// Mitsubishi GX Works2 project: 化成2号柜-5.30   PLC: Q03UDE
// 化成线2号柜

TYPE BarCylinderIO : STRUCT
  xPresentSwitch : BOOL;  (* 行程开关 *)
  xBarCylinder : BOOL;  (* 阻挡气缸 *)
  xEmpty : BOOL;  (* 为空指示 *)
  xTransportMotorCW : BOOL;  (* 输送电机正转 *)
  tLeaveDelay : TIME;  (* 放行延时 *)
  xUnload : BOOL;  (* 下料 *)
  xBarCylinderButton : BOOL;  (* 阻挡气缸 *)
  xTransportMotorCWButton : BOOL;  (* 输送电机正转按钮 *)
  xLoad : BOOL;  (* 上料 *)
  xNextRun : BOOL;  (* 下位设备开始运行 *)
  xTransportMotorCCWButton : BOOL;  (* 输送电机反转按钮 *)
  xTransportMotorCCW : BOOL;  (* 输送电机反转 *)
END_STRUCT END_TYPE

TYPE ConveyorIO : STRUCT
  xCWPresent : BOOL;  (* 正转检测有无传感器 *)
  xCCWPresent : BOOL;  (* 反转检测有无传感器 *)
  xLoad : BOOL;  (* 上料请求 *)
  xUnload : BOOL;  (* 下料请求 *)
  xMotorCW : BOOL;  (* 电机正转 *)
  xMotorCCW : BOOL;  (* 电机反转 *)
  xEmpty : BOOL;  (* 线体状态为空 *)
  xNextRun : BOOL;  (* 下段线体运行 *)
  xUnloadCCW : BOOL;  (* 下料为反转 *)
  xloadCCW : BOOL;  (* 上料为反转 *)
  xLeave : BOOL;  (* 已经离开 *)
  xForward : BOOL;  (* 正转手动 *)
  xBackward : BOOL;  (* 反转手动 *)
  xBusy : BOOL;  (* 工作中 *)
  xPutInto : BOOL;  (* 线体直接投入物料 *)
  xUnloadAlarm : BOOL;  (* 下料报警 *)
  tLoadDelay : TIME;  (* 进入延时设置 *)
  xPosLimit : BOOL;  (* 正限位 *)
  xNegLimit : BOOL;  (* 负限位 *)
  xOverWidthAlarm : BOOL;  (* 超宽报警 *)
  xLimitAlarrm : BOOL;  (* 限位报警 *)
  iDeviceID : INT;  (* 线体ID *)
END_STRUCT END_TYPE

TYPE RGVCommunication : STRUCT
  xFullLoadRequest : BOOL;  (* 满框上料请求 *)
  xFullUnloadRequest : BOOL;  (* 满框下料请求 *)
  xEmptyLoadRequest : BOOL;  (* 空框上料请求 *)
  xEmptyUnloadRequest : BOOL;  (* 空框下料请求 *)
  xFullLoadRequestAkn : BOOL;  (* 满框上料请求确认 *)
  xFullUnloadRequestAkn : BOOL;  (* 满框下料请求确认 *)
  xEmptyLoadRequestAkn : BOOL;  (* 空框上料请求确认 *)
  xEmptyUnloadRequestAkn : BOOL;  (* 空框下料请求确认 *)
  xFullLoadComplete : BOOL;  (* 满框上料完成 *)
  xFullUnloadComplete : BOOL;  (* 满框下料完成 *)
  xEmptyLoadComplete : BOOL;  (* 空框上料完成 *)
  xEmptyUnloadComplete : BOOL;  (* 空框下料完成 *)
  xFullLoadCompleteAkn : BOOL;  (* 满框上料完成确认 *)
  xFullUnloadCompleteAkn : BOOL;  (* 满框下料完成确认 *)
  xEmptyLoadCompleteAkn : BOOL;  (* 空框上料完成确认 *)
  xEmptyUnloadCompleteAkn : BOOL;  (* 空框下料完成确认 *)
  iCurrentPostion : INT;  (* RGV当前位置 *)
  iDestinationPos : INT;  (* RGV目标位置 *)
  xMdiExe : BOOL;  (* RGV 执行 *)
  xMdiDone : BOOL;  (* RGV 执行完成 *)
  xEmpty1 : BOOL;
  xNextRun1 : BOOL;
  xEmpty2 : BOOL;
  xNextRun2 : BOOL;
  xLoad1 : BOOL;
  xUnload1 : BOOL;
  xLoad2 : BOOL;
  xUnload2 : BOOL;
  xCollisionAlarm : BOOL;  (* 干涉报警 *)
  xRemoteReset : BOOL;  (* 远程复位 *)
  xAuto : BOOL;  (* 自动 *)
END_STRUCT END_TYPE

TYPE ShuttleCarIO : STRUCT
  xReady : BOOL;  (* 准备就绪 *)
  xForward : BOOL;  (* 正转 *)
  xBackward : BOOL;  (* 反转 *)
  iCurrentPos : INT;  (* 当前位置 *)
  iDestinationPos : INT;  (* 目标位置 *)
  xCW : BOOL;  (* 正转输出 *)
  xCCW : BOOL;  (* 反转输出 *)
  xBrake : BOOL;  (* 刹车 *)
  xHomeSwitch : BOOL;  (* 零位接近开关 *)
  xPosLimit : BOOL;  (* 正限位 *)
  xNegLimit : BOOL;  (* 负限位 *)
  xMDIExe : BOOL;  (* MDI开始 *)
  xMDIDone : BOOL;  (* MDI 完成 *)
  xPassLimit : BOOL;  (* 限位屏蔽 *)
  xPosLimitCatch : BOOL;  (* 正限位捕捉 *)
  xNegLimitCatch : BOOL;  (* 负限位捕捉 *)
  xHomeExe : BOOL;  (* 开始寻零 *)
  xHomeDone : BOOL;  (* 寻零完成 *)
  xHomeBusy : BOOL;  (* 寻零中 *)
  xHomeFailed : BOOL;  (* 寻零失败 *)
  xBusy : BOOL;  (* 工作中 *)
  tArriveDelay : TIME;  (* 到位延时 *)
  xCylinder : BOOL;  (* 气缸控制 *)
  tBrakeDelay : TIME;  (* 抱闸延时 *)
  xPauseRamp : BOOL;  (* 暂停减速斜坡标志位 *)
  xPresentDetect1 : BOOL;  (* 物料有无检测1 *)
  xPresentDetect2 : BOOL;  (* 物料有无检测2 *)
  xOvertimeAlarm : BOOL;  (* 超时报警 *)
  tSetOverTime : TIME;  (* 设置超时时间 *)
  xLooseDetect : BOOL;  (* 松绳检测 *)
  xLooseAlarm : BOOL;  (* 松绳报警 *)
END_STRUCT END_TYPE

TYPE SwitchIO : STRUCT
  xLiftCylinderRetractDetect : BOOL;
  xLiftCylinderExtendDetect : BOOL;
  xLiftCylinderRetract : BOOL;
  xLiftCylinderExtend : BOOL;
  xEntryBarCylinderRetract : BOOL;
  xLiftCylinderExtendInit : BOOL;
  xEntryEnable : BOOL;
  xExitEnable : BOOL;
  xExitBarCylinderRetract : BOOL;
  xSwithEnable : BOOL;
  xLiftCylinderRetractButton : BOOL;
  xLiftCylinderExtendButton : BOOL;
  xEntryBarCylinderRetractButton : BOOL;
  xExitBarCylinderRetractButton : BOOL;
END_STRUCT END_TYPE

TYPE Stub : STRUCT
  xLoadRequest : BOOL;
  xLoadRequestAkn : BOOL;
  xUnloadRequest : BOOL;
  xUnloadRequestAkn : BOOL;
END_STRUCT END_TYPE

TYPE AccumulateConveyorIO : STRUCT
  xBarCylinderButton : BOOL;  (* 阻挡气缸按钮 *)
  xBarCylinder : BOOL;  (* 阻挡气缸 *)
  xLoad : BOOL;  (* 上料 *)
  xEmpty : BOOL;  (* 为空指示 *)
  xNextRun : BOOL;  (* 下位设备开始运行 *)
  xUnload : BOOL;  (* 下料 *)
  xTransportMotorCWButton : BOOL;  (* 输送电机正转按钮 *)
  xTransportMotorCW : BOOL;  (* 输送电机正转 *)
  xTransportMotorCCWButton : BOOL;  (* 输送电机反转按钮 *)
  xTransportMotorCCW : BOOL;  (* 输送电机反转 *)
  tLeaveDelay : TIME;  (* 放行延时 *)
  xPresentSwitch : BOOL;  (* 行程开关正向 *)
  xPresentSwitchEntry : BOOL;  (* 行程开关反向 *)
  xBarCylinderSecondary : BOOL;  (* 阻挡第二个无料的气缸 *)
  xBarSecondaryButton : BOOL;  (* 阻挡第二个无料的气缸手动按钮 *)
  xTwoWay : BOOL;  (* 双向积放线 *)
  iAccumulate : INT;  (* 数量 *)
  xLoadDone : BOOL;  (* 上料完成 *)
  tLoadDelay : TIME;  (* 上料延时 *)
  iDeviceID : INT;
END_STRUCT END_TYPE

// global labels: Global1
VAR_GLOBAL
  g_xAuto AT M11 : BOOL;  (* 自动 *)
  g_xManual : BOOL;  (* 手动 *)
  g_xEStop AT X3 : BOOL;  (* 急停 *)
  g_xReset AT X0 : BOOL;  (* 复位 *)
  g_xStackLampRed AT Y100 : BOOL;
  g_xStackLampAmber AT Y101 : BOOL;
  g_xStackLampGreen AT Y102 : BOOL;
  g_xBuzzer AT Y103 : BOOL;
  g_xStop AT M2 : BOOL;  (* 停止 *)
  g_xLocalAutoStart AT M1 : BOOL;  (* 本地自动启动 *)
  g_xRemoteAutoStart AT M0 : BOOL;  (* 远程自动启动 *)
  g_xRemoteAuto AT M10 : BOOL;  (* 远程 *)
  g_iState AT D40 : INT;  (* 当前状态 *)
  g_iLocalAutoStep : INT;
  g_xError : BOOL;
  g_xStart : BOOL;  (* 启动 *)
  g_xResetSingle AT M4 : BOOL;  (* 单线体复位 *)
  g_iDeviceIDSelect AT D0 : INT;  (* 线体编号选择 *)
  g_xPause AT M3 : BOOL;  (* 暂停 *)
  g_xAlarm : BOOL;  (* 报警 *)
  g_xInsertTask AT M5 : BOOL;  (* 单线体插入 *)
  g_iInsertTask AT D2 : INT;  (* 插入数据 *)
END_VAR

// global labels: Global
VAR_GLOBAL
  g_xQuarPackageRGVComFailed : BOOL;
  g_xChemRGVComFailed : BOOL;
  g_xChem1ComFailed : BOOL;
END_VAR

// task Task_01 (event TRUE, interval 0, priority 31): Start, POU, UDP

FUNCTION_BLOCK BarCylinder
VAR_IN_OUT
  BarCylinderIO : BarCylinderIO;
END_VAR
VAR
  m_tonViaDelay : TON;  (* 卸料延时定时器 *)
  m_xViaDelay : BOOL;  (* 通过延时 *)
  m_tViaDelayElapse : TIME;  (* 通过延时当前时间 *)
  m_xInitial : BOOL;  (* 初始化 *)
END_VAR
  (***********************************************************************
阻挡器模块，
由一个行程开关，一个阻挡器，一个倍速链输送电机组成
具有手动与自动模式
xEmpty显示当前为空料的状态
xUnload为卸料信号，连接下一设备的xEmpty信号
*************************************************************************)

  (*初始化，离开延时时间设置为5秒*)
IF NOT m_xInitial THEN
	 BarCylinderIO.tLeaveDelay :=T#5s;
	m_xInitial:=1;
END_IF;
IF g_xManual THEN    (*手动*)
	BarCylinderIO.xNextRun:=0;
	IF BarCylinderIO.xBarCylinderButton THEN
		BarCylinderIO.xBarCylinder:=1;
	ELSE
		BarCylinderIO.xBarCylinder:=0;
	END_IF;
	IF BarCylinderIO.xTransportMotorCWButton 
		AND NOT BarCylinderIO.xTransportMotorCCWButton 
		AND NOT BarCylinderIO.xTransportMotorCCW   THEN
		BarCylinderIO.xTransportMotorCW:=1;
	ELSE
		BarCylinderIO.xTransportMotorCW:=0;
	END_IF;
	IF BarCylinderIO.xTransportMotorCCWButton 
		AND NOT BarCylinderIO.xTransportMotorCWButton 
		AND NOT BarCylinderIO.xTransportMotorCW   THEN
		BarCylinderIO.xTransportMotorCCW:=1;
	ELSE
		BarCylinderIO.xTransportMotorCCW:=0;
	END_IF;
END_IF;
(*离开延时定时器*)
m_tonViaDelay(IN:=NOT  BarCylinderIO.xPresentSwitch AND g_xAuto  ,PT:= BarCylinderIO.tLeaveDelay ,Q:= BarCylinderIO.xEmpty ,ET:=m_tViaDelayElapse );

IF g_xAuto THEN(*自动*)
    IF BarCylinderIO.xUnload  AND NOT BarCylinderIO.xEmpty AND NOT BarCylinderIO.xNextRun THEN(*收到卸料命令，当阻挡器不为空时*)
    	BarCylinderIO.xBarCylinder:=1;
    	BarCylinderIO.xNextRun:=1;(*确保下料命令只执行一次，防止物料在输送过程中又有卸料命令导致多事卸料*)
    	BarCylinderIO.xTransportMotorCW:=1;
    END_IF;
    IF NOT  BarCylinderIO.xUnload  THEN
    	BarCylinderIO.xNextRun:=0;
    END_IF;
    (*如果为空，气缸顶起*)
   IF  BarCylinderIO.xEmpty  THEN
   	   BarCylinderIO.xBarCylinder:=0;
   	   IF BarCylinderIO.xLoad THEN
	   	   BarCylinderIO.xTransportMotorCW:=1;
	   END_IF;
   END_IF;
   IF NOT BarCylinderIO.xUnload AND NOT  BarCylinderIO.xEmpty THEN
   	    BarCylinderIO.xTransportMotorCW:=0;
   	END_IF;
END_IF;
IF NOT g_xEStop THEN
	 BarCylinderIO.xTransportMotorCW:=0;
	 BarCylinderIO.xTransportMotorCCW:=0;
	 BarCylinderIO.xBarCylinder:=0;
END_IF;
END_FUNCTION_BLOCK

FUNCTION_BLOCK Conveyor
VAR
  tRundelay : TIME;  (* 离开延时 *)
END_VAR
VAR_IN_OUT
  ConveyorMotor : ConveyorIO;  (* 输送线输入输出 *)
END_VAR
VAR
  iStep : INT;  (* 上料步骤 *)
  m_tUnloadTimer : TIME;  (* 下料计时器 *)
  m_tonLeaveDelay : TON;  (* 离开延时定时器 *)
  m_xLeaveDelayOut : BOOL;  (* 离开延时 *)
  m_tLeaveCurrentTime : TIME;
END_VAR
VAR CONSTANT
  LOAD_UNLOAD_TIME : TIME := T#30s;  (* 延时报警常量 *)
END_VAR
VAR
  m_tonUnloadAlam : TON;  (* 下料报警定时器 *)
  m_tonLoadDelay : TON;  (* 离开延时定时器 *)
  m_xLoadDelayOut : BOOL;  (* 离开延时 *)
  m_tLoadCurrentTime : TIME;
  m_xInitial : BOOL;  (* 初始化 *)
  m_tLoadTimer : TIME;  (* 上料延时当前时间 *)
END_VAR
(*////////////////////////////////////////////////////////////////////////////////////////////////////////////
//传输线控制FB块，可控制单方向线体，双向旋转线体，支持双向上下料            
//线体初始化后为空的情况下输入xLoad信号即可进行上料动作，使用xLoadCCW信号可反方向上料
//增加了产品信息和产品种类的储存，当传输线为空和上料进行标志位为零的情况下清除产品信息和产品种类
//使用方式是在置位xLoad信号后，把产品信息和产品种类传入，等下料后自动清零
//线体不为空的情况下使用xUnload信号可进行下料动作，物料有无传感器的下降沿后出发计时器，延时断开传输线旋转
//单方向传输线体把xLoadCCW、xUnloadCCW设置为零，双向线体上料方向和下料反向的,方向固定的 把xUnloadCCW设置为1
//双方向线体双向都能上下料的要根据上料的方向来设置xLoadCCW,xUnloadCCW
//增加工作中信号xBusy当电机正转 显示为工作中
//增加上下料超时报警，xLoadAlarm，xUnloadAlarm，设定时间在LOAD_UNLOAD_TIME常量上，现在设置的为30秒
//增加xPutInto信号，用于直接投入的物料，检测开关感应到后，直接进入下料流程，上升沿有效
//离开延时改为变量 iLeaveDelay 默认为0 离开检测开关离输送线尾端比较远的线体需要根据情况设定100ms为单位
增加初始化标志位，增加进入延时时间，初始化为进入延时时间为0 ，离开延时时间为2S，通过外围接口可以更改
//修改信息  修改后请增加版本
//YAO      V1.0
///////////////////////////////////////////////////////////////////////////////////////////////////////////
********************************************************)
IF NOT m_xInitial THEN
	ConveyorMotor.tLoadDelay:=T#100ms;
	ConveyorMotor.xNegLimit:=1;
	ConveyorMotor.xPosLimit:=1;
END_IF;
m_xInitial:=1;
IF g_xAuto THEN
CASE iStep OF
	0:
	ConveyorMotor.xMotorCW:=0;
	ConveyorMotor.xMotorCCW:=0;
	ConveyorMotor.xNextRun:=0;
IF g_xEStop AND NOT ConveyorMotor.xLimitAlarrm  THEN
	IF (ConveyorMotor.xCWPresent OR ConveyorMotor.xCCWPresent)  THEN
		iStep:=3;
		ConveyorMotor.xEmpty:=0;
		ELSE
		iStep:=1;
		ConveyorMotor.xEmpty:=1;
	END_IF;
END_IF;		
	1: 
	IF ConveyorMotor.xLoad    
		AND ConveyorMotor.xMotorCW=0   
		AND ConveyorMotor.xMotorCCW=0   
		AND ConveyorMotor.xEmpty THEN	
		iStep:=2;
	END_IF;
	2: 
	IF ConveyorMotor.xloadCCW THEN
		ConveyorMotor.xMotorCCW:=1; 
		ConveyorMotor.xMotorCW:=0;
	ELSE
	    ConveyorMotor.xMotorCW:=1;  
		ConveyorMotor.xMotorCCW:=0;
	END_IF;
		m_tonLoadDelay(IN:= (ConveyorMotor.xCWPresent AND NOT ConveyorMotor.xloadCCW) 
		                                        OR (ConveyorMotor.xCCWPresent AND ConveyorMotor.xloadCCW) ,
		                               PT:= ConveyorMotor.tLoadDelay ,
		                               Q:= m_xLoadDelayOut ,
		                               ET:= m_tLoadTimer );
	    IF m_xLoadDelayOut THEN 	 
		    iStep:=3;
		END_IF;
	3:
	ConveyorMotor.xMotorCW:=0;
	ConveyorMotor.xMotorCCW:=0;
	ConveyorMotor.xEmpty:=0;
	IF ConveyorMotor.xUnload AND NOT ConveyorMotor.xOverWidthAlarm THEN 
		iStep:=4;
	END_IF;
	4:	
	IF ConveyorMotor.xUnloadCCW THEN   
		ConveyorMotor.xMotorCCW:=1;  
		ConveyorMotor.xMotorCW:=0;
		ELSE
	    ConveyorMotor.xMotorCW:=1;  
		ConveyorMotor.xMotorCCW:=0;
	END_IF;
	ConveyorMotor.xNextRun:=1; 
	IF NOT ConveyorMotor.xUnload THEN 
		istep:=0;
	END_IF;
END_CASE;
IF LDP(TRUE,ConveyorMotor.xPutInto) THEN
	iStep:=0;
END_IF;
END_IF;
IF g_xManual THEN
	iStep:=0;

	IF ConveyorMotor.xForward 
		AND ConveyorMotor.xBackward=0 
		AND ConveyorMotor.xMotorCCW=0
		AND g_xEStop THEN
		ConveyorMotor.xMotorCW:=1;
		ConveyorMotor.xMotorCCW:=0;
		ELSE
		ConveyorMotor.xMotorCW:=0;
	END_IF;

	IF ConveyorMotor.xBackward 
		AND ConveyorMotor.xForward=0 
		AND ConveyorMotor.xMotorCW=0
		AND g_xEStop  THEN
		ConveyorMotor.xMotorCCW:=1;
		conveyormotor.xMotorCW:=0;
		ELSE
		ConveyorMotor.xMotorCCW:=0;
	END_IF;
END_IF;
IF ConveyorMotor.xMotorCCW        
	OR ConveyorMotor.xMotorCW THEN  
	ConveyorMotor.xBusy:=1;
	ELSE
	ConveyorMotor.xBusy:=0;
END_IF;
m_tonUnloadAlam(IN:= iStep=4,PT:= LOAD_UNLOAD_TIME,Q:= ConveyorMotor.xUnloadAlarm,ET:= m_tUnloadTimer );
(*//复位*)
IF (*g_xReset OR*)
	 (g_xResetSingle AND ConveyorMotor.iDeviceID=g_iDeviceIDSelect)THEN (*AND ConveyorMotor.iDeviceID=g_iDeviceIDSelect  THEN*)  (* //非正常情况下切断xNextRun不会复位，通过这个标志位会出发报警*)(*增加单体复位*)
	iStep:=0;
	ConveyorMotor.xNextRun:=0; 
	ConveyorMotor.xLimitAlarrm:=0;
	ConveyorMotor.xOverWidthAlarm:=0;
END_IF;
IF iStep=3 AND (NOT ConveyorMotor.xNegLimit OR NOT ConveyorMotor.xPosLimit) THEN
	ConveyorMotor.xOverWidthAlarm:=1;
END_IF;
IF ( ((ConveyorMotor.xloadCCW AND NOT ConveyorMotor.xNegLimit)            (*反转上料，碰到负限位*)
	OR  ( NOT ConveyorMotor.xloadCCW AND NOT ConveyorMotor.xPosLimit)) (*正转上料，碰到正限位*)
    AND iStep=2) (*上料过程*)
    OR
   ( iStep=4 (*下料过程*)
	AND( (ConveyorMotor.xUnloadCCW AND NOT ConveyorMotor.xPosLimit)  
	OR (NOT ConveyorMotor.xUnloadCCW AND NOT ConveyorMotor.xNegLimit)))    
    THEN
    ConveyorMotor.xLimitAlarrm:=1;
    iStep:=0;
END_IF;
END_FUNCTION_BLOCK

PROGRAM POU
VAR
  Lifter3 : ShuttleCar;
  Lifter3IO : ShuttleCarIO;
  H3000Conveyor11 : Conveyor;
  H3000Conveyor11IO : ConveyorIO;
  H3000Conveyor12 : Conveyor;
  H3000Conveyor12IO : ConveyorIO;
  H3000Conveyor13 : Conveyor;
  H3000Conveyor13IO : ConveyorIO;
  H3000Conveyor14 : Conveyor;
  H3000Conveyor14IO : ConveyorIO;
  H3000Conveyor15 : Conveyor;
  H3000Conveyor15IO : ConveyorIO;
  H3000Conveyor16 : Conveyor;
  H3000Conveyor16IO : ConveyorIO;
  H3000Conveyor17 : Conveyor;
  H3000Conveyor17IO : ConveyorIO;
  H3000Conveyor18 : Conveyor;
  H3000Conveyor18IO : ConveyorIO;
  H3000Conveyor19 : Conveyor;
  H3000Conveyor19IO : ConveyorIO;
  H3000Conveyor20 : Conveyor;
  H3000Conveyor20IO : ConveyorIO;
  H3000Conveyor21 : Conveyor;
  H3000Conveyor21IO : ConveyorIO;
  H3000Conveyor22 : Conveyor;
  H3000Conveyor22IO : ConveyorIO;
  H2200Conveyor13 : Conveyor;
  H2200Conveyor13IO : ConveyorIO;
  H2200Conveyor14 : Conveyor;
  H2200Conveyor14IO : ConveyorIO;
  H2200Conveyor15 : Conveyor;
  H2200Conveyor15IO : ConveyorIO;
  H2200Conveyor16 : Conveyor;
  H2200Conveyor16IO : ConveyorIO;
  H2200Conveyor17 : Conveyor;
  H2200Conveyor17IO : ConveyorIO;
  H2200Conveyor18 : Conveyor;
  H2200Conveyor18IO : ConveyorIO;
  H2200Conveyor19 : Conveyor;
  H2200Conveyor19IO : ConveyorIO;
  H2200Conveyor20 : Conveyor;
  H2200Conveyor20IO : ConveyorIO;
  H2200Conveyor21 : Conveyor;
  H2200Conveyor21IO : ConveyorIO;
  H2200Conveyor22 : Conveyor;
  H2200Conveyor22IO : ConveyorIO;
  H1000Conveyor11 : Conveyor;
  H1000Conveyor11IO : ConveyorIO;
  H1000Conveyor12 : Conveyor;
  H1000Conveyor12IO : ConveyorIO;
  H1000Conveyor13 : Conveyor;
  H1000Conveyor13IO : ConveyorIO;
  H1000Conveyor14 : Conveyor;
  H1000Conveyor14IO : ConveyorIO;
  H1000Conveyor15 : Conveyor;
  H1000Conveyor15IO : ConveyorIO;
  H1000Conveyor16 : Conveyor;
  H1000Conveyor16IO : ConveyorIO;
  H1000Conveyor19 : Conveyor;
  H1000Conveyor19IO : ConveyorIO;
  H1000Conveyor20 : Conveyor;
  H1000Conveyor20IO : ConveyorIO;
  Conveyor3 : Conveyor;
  Conveyor3IO : ConveyorIO;
  Lifter4 : ShuttleCar;
  Lifter4IO : ShuttleCarIO;
  Conveyor4 : Conveyor;
  Conveyor4IO : ConveyorIO;
  Lifter5 : ShuttleCar;
  Lifter5IO : ShuttleCarIO;
  Conveyor5 : Conveyor;
  Conveyor5IO : ConveyorIO;
  H850Conveyor1 : Conveyor;
  H850Conveyor1IO : ConveyorIO;
  H850Conveyor2 : Conveyor;
  H850Conveyor2IO : ConveyorIO;
  H2200Conveyor1 : Conveyor;
  H2200Conveyor1IO : ConveyorIO;
  ShuttleCar1 : ShuttleCar;
  ShuttleCar1IO : ShuttleCarIO;
  ConveyorShuttleCar : Conveyor;
  ConveyorShuttleCarIO : ConveyorIO;
  H1000Rotor1 : ShuttleCar;
  H1000Rotor1IO : ShuttleCarIO;
  H1000Rotor2 : ShuttleCar;
  H1000Rotor2IO : ShuttleCarIO;
  H1000Rotor1Cylinder : ShuttleCar;
  H1000Rotor1CylinderIO : ShuttleCarIO;
  H1000Rotor2Cylinder : ShuttleCar;
  H1000Rotor2CylinderIO : ShuttleCarIO;
  H850Conveyor1Trans : Conveyor;  (* 二封设备入口接驳 *)
  H850Conveyor1IOTrans : ConveyorIO;  (* 二封设备入口接驳 *)
  H850Conveyor2Trans : Conveyor;  (* 二封设备入口接驳 *)
  H850Conveyor2IOTrans : ConveyorIO;  (* 二封设备入口接驳 *)
  H850Conveyor3Trans : Conveyor;  (* 二封设备入口接驳 *)
  H850Conveyor3IOTrans : ConveyorIO;  (* 二封设备入口接驳 *)
  H850Conveyor4Trans : Conveyor;  (* 二封设备入口接驳 *)
  H850Conveyor4IOTrans : ConveyorIO;  (* 二封设备入口接驳 *)
  H850Conveyor5Trans : Conveyor;  (* 二封设备入口接驳 *)
  H850Conveyor5IOTrans : ConveyorIO;  (* 二封设备入口接驳 *)
  H850Conveyor6Trans : Conveyor;  (* 二封设备入口接驳 *)
  H850Conveyor6IOTrans : ConveyorIO;  (* 二封设备入口接驳 *)
  H850Conveyor7Trans : Conveyor;  (* 二封设备入口接驳 *)
  H850Conveyor7IOTrans : ConveyorIO;  (* 二封设备入口接驳 *)
  H850Conveyor8Trans : Conveyor;  (* 二封设备入口接驳 *)
  H850Conveyor8IOTrans : ConveyorIO;  (* 二封设备入口接驳 *)
  Lifter4VelocityCtl : ShuttleCarVelocityFB;
  Lifter5VelocityCtl : ShuttleCarVelocityFB;
  m_tofShuttleCar1LeaveDelay : TOF;  (* f *)
  m_xShuttleCar1LeaveDelay : BOOL;
  m_tShuttleCar1LeaveDelay : TIME;
  Lifter3VelocityCtl : ShuttleCarVelocityFB;
  H380EmptyABumperBar : AccumulateConveyor;
  H380EmptyABumperBarIO : AccumulateConveyorIO;
  H380EmptyBBumperBar : AccumulateConveyor;
  H380EmptyBBumperBarIO : AccumulateConveyorIO;
  ChemRGV : RGVCommunication;
  QuarPackageRGV : RGVCommunication;
  m_iH1000Rotor2Step : INT;
  m_iH1000Rotor1Step : INT;
  QuarPackage1Stub : Stub;
  QuarPackage2Stub : Stub;
  QuarPackage3Stub : Stub;
  QuarPackage4Stub : Stub;
  Chem1Stub : Stub;
  Chem2Stub : Stub;
  Chem3Stub : Stub;
  Chem4Stub : Stub;
  Chem5Stub : Stub;
  Chem6Stub : Stub;
  Chem7Stub : Stub;
  Chem8Stub : Stub;
  Chem9Stub : Stub;
  Chem10Stub : Stub;
  Chem11Stub : Stub;
  Chem12Stub : Stub;
  m_tonXD8 : TON;
  m_xXD8 : BOOL;
  m_tXD8 : TIME;
  m_xXD8Lock : BOOL;
  m_xDirection : BOOL;  (* 空框方向信息 *)
  m_xRotor2Done : BOOL;  (* 上料转台旋转完成 *)
  m_xRotor1Done : BOOL;  (* 下料转台旋转完成 *)
  m_xRotor1Start : BOOL;  (* 下料转台旋转开始 *)
  m_xRotor2Start : BOOL;  (* 上料转台旋转开始 *)
  m_xDischargeAkn : BOOL;  (* 下料确认 *)
  m_xFomationRGVAuto : BOOL;
  m_xDebindCode : BOOL;
  m_xCheckDone : BOOL;  (* 品检完成 *)
  m_xAllCheck : BOOL;  (* 全检工位 *)
  m_xAllCheckOver : BOOL;  (* 全检完毕按钮 *)
  m_xPassAllow : BOOL;  (* 全检放行 *)
  m_arrxRGVEmptyTaskCondition : ARRAY [0..9] OF BOOL;  (* 空框回流任务 *)
  RGVEmptyTask : PriorityFB;
  m_iRGVEmptyTask : INT;
  H380EmptyBRotorConveyorIO : ConveyorIO;
  H380EmptyBLifter : ShuttleCar;  (* 空框B转台升降气缸 *)
  H380EmptyBLifterIO : ShuttleCarIO;
  H380EmptyBRotor : ShuttleCar;  (* 空框B转台 *)
  H380EmptyBRotorIO : ShuttleCarIO;
  m_xEmptyBRotorStart : BOOL;  (* 空框B旋转开始 *)
  m_xEmptyBRotorDone : BOOL;  (* 空框B旋转完毕 *)
  m_iEmptyBRotorStep : INT;  (* 空框B旋转步 *)
  m_xLoadDirection : BOOL;  (* 上料口方向信息 *)
  m_xUnloadDirection : BOOL;  (* 下料口方向信息 *)
  H380EmptyBRotorConveyor : Conveyor;  (* 空框B转台Conveyor *)
  H380EmptyARotorConveyor : Conveyor;  (* 空框A转台Conveyor *)
  H380EmptyARotorConveyorIO : ConveyorIO;
  H380EmptyALifter : ShuttleCar;  (* 空框A转台升降气缸 *)
  H380EmptyALifterIO : ShuttleCarIO;
  H380EmptyARotor : ShuttleCar;  (* 空框A转台 *)
  H380EmptyARotorIO : ShuttleCarIO;
  m_xEmptyARotorStart : BOOL;  (* 空框A旋转开始 *)
  m_xEmptyARotorDone : BOOL;  (* 空框A旋转完毕 *)
  m_iEmptyARotorStep : INT;  (* 空框A旋转步 *)
  TON_BRotorStep5 : TON;  (* 空框B转台第5步计时 *)
  m_xBRotorStep5 : BOOL;
  m_tBRotorStep5 : TIME;
  TON_ARotorStep5 : TON;  (* 空框A转台第5步延时 *)
  m_xARotorStep5 : BOOL;
  m_tARotorStep5 : TIME;
  H2200SudsecitonCylinderA3 : BarCylinder;  (* 空框回流A线3阻挡气缸 *)
  H2200SudsecitonCylinderA4 : BarCylinder;  (* 空框回流A线4阻挡气缸 *)
  H2200SudsecitonCylinderA5 : BarCylinder;  (* 空框回流A线5阻挡气缸 *)
  H2200SudsecitonCylinderA3IO : BarCylinderIO;  (* 空框回流A线3阻挡气缸 *)
  H2200SudsecitonCylinderA4IO : BarCylinderIO;  (* 空框回流A线4阻挡气缸 *)
  H2200SudsecitonCylinderA5IO : BarCylinderIO;  (* 空框回流A线5阻挡气缸 *)
  H2200SudsecitonCylinderB3 : BarCylinder;  (* 空框回流B线3阻挡气缸 *)
  H2200SudsecitonCylinderB4 : BarCylinder;  (* 空框回流B线4阻挡气缸 *)
  H2200SudsecitonCylinderB5 : BarCylinder;  (* 空框回流B线5阻挡气缸 *)
  H2200SudsecitonCylinderB3IO : BarCylinderIO;  (* 空框回流B线3阻挡气缸 *)
  H2200SudsecitonCylinderB4IO : BarCylinderIO;  (* 空框回流B线4阻挡气缸 *)
  H2200SudsecitonCylinderB5IO : BarCylinderIO;  (* 空框回流B线5阻挡气缸 *)
  m_tonSudsecitonCylinderA3Delay : TON;  (* 空框回流A线5阻挡气缸 *)
  m_tCylinderA3DelayCurrentTime : TIME;
  m_tonSudsecitonCylinderA4Delay : TON;
  m_tCylinderA4DelayCurrentTime : TIME;
  m_tonSudsecitonCylinderA5Delay : TON;
  m_tCylinderA5DelayCurrentTime : TIME;
  m_tonSudsecitonCylinderB3Delay : TON;
  m_tCylinderB3DelayCurrentTime : TIME;
  m_tonSudsecitonCylinderB4Delay : TON;
  m_tCylinderB4DelayCurrentTime : TIME;
  m_tonSudsecitonCylinderB5Delay : TON;
  m_tCylinderB5DelayCurrentTime : TIME;
  BlockA : BOOL;  (* 空框回流A线阻塞 *)
  BlockB : BOOL;  (* 空框回流B线阻塞 *)
END_VAR
(*---------我在516行加了一整行*)
Lifter3(ShuttleCarInOut:=Lifter3IO);
ShuttleCarCurrentPosition( X5A OR X5B ,X5A ,X5B, FALSE, Lifter3IO.iCurrentPos );
Lifter3VelocityCtl(xEnable:= g_xManual,xMotorCW:= Lifter3IO.xCW ,xMotorCCW:= Lifter3IO.xCCW ,
                               xPosition1Switch:= X5A ,xDecelerationSwitch:= X59 ,
	                           xPosition2Switch:=X5B ,xHighSpeed:= Y163);
Lifter3IO.xReady:=X4;
Lifter3Io.xForward:=M50;
Lifter3IO.xBackward:=M51;
Lifter3IO.xPosLimit:=X5C;
Lifter3IO.xNegLimit:=X5D;
Lifter3Io.xLooseDetect:=X5E;
M130:=Lifter3IO.xLooseDetect;
Y161:=Lifter3IO.xCW;
Y162:=Lifter3IO.xCCW;
Y166:=Lifter3IO.xBrake;

Conveyor3(ConveyorMotor:=Conveyor3IO);
Conveyor3IO.xForward:=M52;
Conveyor3IO.xBackward:=M53;
Conveyor3IO.xCWPresent:=X61;
Conveyor3IO.xCCWPresent:=X62;
Y168:=Conveyor3IO.xMotorCW;
Y167:=Conveyor3IO.xMotorCCW;
Conveyor3IO.xUnloadCCW:=1;
Conveyor3IO.iDeviceID:=3;

Lifter4(ShuttleCarInOut:=Lifter4IO);
ShuttleCarCurrentPosition( X64 OR X65 ,X64 ,X65, FALSE, Lifter4IO.iCurrentPos );
Lifter4VelocityCtl(xEnable:= g_xAuto,xMotorCW:= Lifter4IO.xCW ,xMotorCCW:= Lifter4IO.xCCW ,
                               xPosition1Switch:= X64 ,xDecelerationSwitch:= X63 ,
	                           xPosition2Switch:=X65 ,xHighSpeed:= Y16B);
Lifter4IO.xReady:=X5;
Lifter4Io.xForward:=M54;
Lifter4IO.xBackward:=M55;
Lifter4IO.xPosLimit:=X66;
Lifter4IO.xNegLimit:=X67;
Lifter4IO.xLooseDetect:=X68;
M129:=Lifter4IO.xLooseAlarm;
Y169:=Lifter4IO.xCW;
Y16A:=Lifter4IO.xCCW;
Y16E:=Lifter4IO.xBrake;

Conveyor4(ConveyorMotor:=Conveyor4IO);
Conveyor4IO.xForward:=M56;
Conveyor4IO.xBackward:=M57;
Conveyor4IO.xCWPresent:=X6B;
Conveyor4IO.xCCWPresent:=X6C;
Y170:=Conveyor4IO.xMotorCW;
Y16F:=Conveyor4IO.xMotorCCW;
Conveyor4IO.xUnloadCCW:=1;
Conveyor4IO.iDeviceID:=4;

Lifter5(ShuttleCarInOut:=Lifter5IO);
ShuttleCarCurrentPosition( X6E OR X6F ,X6E ,X6F, FALSE, Lifter5IO.iCurrentPos );
Lifter5VelocityCtl(xEnable:= g_xAuto,
                               xMotorCW:= Lifter5IO.xCW ,
                               xMotorCCW:= Lifter5IO.xCCW,
                               xPosition1Switch:=X6E,
                               xDecelerationSwitch:= X6D,
	                           xPosition2Switch:=X6F,
	                           xHighSpeed:= Y173 );
Lifter5IO.xReady:=X6;
Lifter5Io.xForward:=M58;
Lifter5IO.xBackward:=M59;
Lifter5IO.xPosLimit:=X70;
Lifter5IO.xNegLimit:=X71;
Lifter5IO.xLooseDetect:=X72;
M128:=Lifter5IO.xLooseAlarm;
Y171:=Lifter5IO.xCW;
Y172:=Lifter5IO.xCCW;
Y176:=Lifter5IO.xBrake;

Conveyor5(ConveyorMotor:=Conveyor5IO);
Conveyor5IO.xForward:=M60;
Conveyor5IO.xBackward:=M61;
Conveyor5IO.xCWPresent:=X75;
Conveyor5IO.xCCWPresent:=X76;
Y178:=Conveyor5IO.xMotorCW;
Y177:=Conveyor5IO.xMotorCCW;
Conveyor5IO.xUnloadCCW:=1;
Conveyor5IO.iDeviceID:=5;

ShuttleCar1(ShuttleCarInOut:=ShuttleCar1IO);
ShuttleCarCurrentPosition(( NOT X53 AND NOT X54) OR (NOT X53 AND NOT X55) OR (NOT X54 AND NOT  X55) ,
                                                       NOT X53 AND NOT X54 ,
                                                       NOT X53 AND NOT X55,
                                                       NOT X54 AND NOT  X55, 
                                                       ShuttleCar1IO.iCurrentPos );
ShuttleCar1IO.xReady:=X7;
ShuttleCar1IO.xForward:=M62;
ShuttleCar1IO.xBackward:=M63;
ShuttleCar1IO.xPosLimit:=X51;
ShuttleCar1IO.xNegLimit:=X52;
Y1AC:=ShuttleCar1IO.xCW;
Y1AB:=ShuttleCar1IO.xCCW;
Y12B:=ShuttleCar1IO.xBrake;

ConveyorShuttleCar(ConveyorMotor:=ConveyorShuttleCarIO);
ConveyorShuttleCarIO.xForward:=M64;
ConveyorShuttleCarIO.xBackward:=M65;
ConveyorShuttleCarIO.xCWPresent:=X56;
ConveyorShuttleCarIO.xCCWPresent:=X57;
Y153:=ConveyorShuttleCarIO.xMotorCW;
Y154:=ConveyorShuttleCarIO.xMotorCCW;
ConveyorShuttleCarIO.iDeviceID:=6;

H3000Conveyor11(ConveyorMotor:=H3000Conveyor11IO);
H3000Conveyor11IO.xForward:=M30;
H3000Conveyor11IO.xCWPresent:=X8;
Y108:=H3000Conveyor11IO.xMotorCW;
H3000Conveyor11IO.iDeviceID:=3011;

H3000Conveyor12(ConveyorMotor:=H3000Conveyor12IO);
H3000Conveyor12IO.xForward:=M31;
H3000Conveyor12IO.xCWPresent:=X9;
Y109:=H3000Conveyor12IO.xMotorCW;
H3000Conveyor12IO.iDeviceID:=3012;

H3000Conveyor13(ConveyorMotor:=H3000Conveyor13IO);
H3000Conveyor13IO.xForward:=M32;
H3000Conveyor13IO.xCWPresent:=XA;
Y10A:=H3000Conveyor13IO.xMotorCW;
H3000Conveyor13IO.iDeviceID:=3013;

H3000Conveyor14(ConveyorMotor:=H3000Conveyor14IO);
H3000Conveyor14IO.xForward:=M33;
H3000Conveyor14IO.xCWPresent:=XB;
Y10B:=H3000Conveyor14IO.xMotorCW;
H3000Conveyor14IO.iDeviceID:=3014;

H3000Conveyor15(ConveyorMotor:=H3000Conveyor15IO);
H3000Conveyor15IO.xForward:=M34;
H3000Conveyor15IO.xCWPresent:=XC;
Y10C:=H3000Conveyor15IO.xMotorCW;
H3000Conveyor15IO.iDeviceID:=3015;

H3000Conveyor16(ConveyorMotor:=H3000Conveyor16IO);
H3000Conveyor16IO.xForward:=M34;
H3000Conveyor16IO.xCWPresent:=XD;
Y10D:=H3000Conveyor16IO.xMotorCW;
H3000Conveyor16IO.iDeviceID:=3016;

H3000Conveyor17(ConveyorMotor:=H3000Conveyor17IO);
H3000Conveyor17IO.xForward:=M35;
H3000Conveyor17IO.xCWPresent:=XE;
Y10E:=H3000Conveyor17IO.xMotorCW;
H3000Conveyor17IO.iDeviceID:=3017;

H3000Conveyor18(ConveyorMotor:=H3000Conveyor18IO);
H3000Conveyor18IO.xForward:=M36;
H3000Conveyor18IO.xCWPresent:=XF;
Y10F:=H3000Conveyor18IO.xMotorCW;
H3000Conveyor18IO.iDeviceID:=3018;

H3000Conveyor19(ConveyorMotor:=H3000Conveyor19IO);
H3000Conveyor19IO.xForward:=M37;
H3000Conveyor19IO.xCWPresent:=X10;
Y110:=H3000Conveyor19IO.xMotorCW;
H3000Conveyor19IO.iDeviceID:=3019;

H3000Conveyor20(ConveyorMotor:=H3000Conveyor20IO);
H3000Conveyor20IO.xForward:=M38;
H3000Conveyor20IO.xCWPresent:=X11;
Y111:=H3000Conveyor20IO.xMotorCW;
H3000Conveyor20IO.iDeviceID:=3020;

H3000Conveyor21(ConveyorMotor:=H3000Conveyor21IO);
H3000Conveyor21IO.xForward:=M39;
H3000Conveyor21IO.xCWPresent:=X12;
Y112:=H3000Conveyor21IO.xMotorCW;
H3000Conveyor21IO.iDeviceID:=3021;

H3000Conveyor22(ConveyorMotor:=H3000Conveyor22IO);
H3000Conveyor22IO.xForward:=M40;
H3000Conveyor22IO.xCWPresent:=X13;
Y113:=H3000Conveyor22IO.xMotorCW;
H3000Conveyor22IO.xNegLimit:=X14;
M98:=H3000Conveyor22IO.xOverWidthAlarm;
M99:=H3000Conveyor22IO.xLimitAlarrm;
H3000Conveyor22IO.iDeviceID:=3022;

H850Conveyor1(ConveyorMotor:=H850Conveyor1IO);
H850Conveyor1IO.xForward:=M41;
H850Conveyor1IO.xCWPresent:=X4E;
Y14E:=H850Conveyor1IO.xMotorCW;
H850Conveyor1IO.iDeviceID:=8501;

H850Conveyor2(ConveyorMotor:=H850Conveyor2IO);
H850Conveyor2IO.xForward:=M42;
H850Conveyor2IO.xCWPresent:=X4F;
Y14F:=H850Conveyor2IO.xMotorCW;
H850Conveyor2IO.iDeviceID:=8502;

H2200Conveyor1(ConveyorMotor:=H2200Conveyor1IO);
H2200Conveyor1IO.xForward:=M43;
H2200Conveyor1IO.xCWPresent:=X4D;
Y14D:=H2200Conveyor1IO.xMotorCW;
H2200Conveyor1IO.iDeviceID:=2201;


H2200Conveyor13(ConveyorMotor:=H2200Conveyor13IO);
H2200Conveyor13IO.xForward:=M44;
H2200Conveyor13IO.xCWPresent:=X2F;
Y12F:=H2200Conveyor13IO.xMotorCW;
H2200Conveyor13IO.iDeviceID:=2213;

H2200Conveyor14(ConveyorMotor:=H2200Conveyor14IO);
H2200Conveyor14IO.xForward:=M45;
H2200Conveyor14IO.xCWPresent:=X30;
Y130:=H2200Conveyor14IO.xMotorCW;
H2200Conveyor14IO.iDeviceID:=2214;

H2200Conveyor15(ConveyorMotor:=H2200Conveyor15IO);
H2200Conveyor15IO.xForward:=M46;
H2200Conveyor15IO.xCWPresent:=X31;
Y131:=H2200Conveyor15IO.xMotorCW;
H2200Conveyor15IO.iDeviceID:=2215;

H2200Conveyor16(ConveyorMotor:=H2200Conveyor16IO);
H2200Conveyor16IO.xForward:=M47;
H2200Conveyor16IO.xCWPresent:=X32;
Y132:=H2200Conveyor16IO.xMotorCW;
H2200Conveyor16IO.iDeviceID:=2216;

H2200Conveyor17(ConveyorMotor:=H2200Conveyor17IO);
H2200Conveyor17IO.xForward:=M48;
H2200Conveyor17IO.xCWPresent:=X33;
Y133:=H2200Conveyor17IO.xMotorCW;
H2200Conveyor17IO.iDeviceID:=2217;

H2200Conveyor18(ConveyorMotor:=H2200Conveyor18IO);
H2200Conveyor18IO.xForward:=M49;
H2200Conveyor18IO.xCWPresent:=X34;
Y134:=H2200Conveyor18IO.xMotorCW;
H2200Conveyor18IO.iDeviceID:=2218;

H2200Conveyor19(ConveyorMotor:=H2200Conveyor19IO);
H2200Conveyor19IO.xForward:=M70;
H2200Conveyor19IO.xCWPresent:=X35;
Y135:=H2200Conveyor19IO.xMotorCW;
H2200Conveyor19IO.iDeviceID:=2219;

H2200Conveyor20(ConveyorMotor:=H2200Conveyor20IO);
H2200Conveyor20IO.xForward:=M71;
H2200Conveyor20IO.xCWPresent:=X36;
Y136:=H2200Conveyor20IO.xMotorCW;
H2200Conveyor20IO.iDeviceID:=2220;

H2200Conveyor21(ConveyorMotor:=H2200Conveyor21IO);
H2200Conveyor21IO.xForward:=M72;
H2200Conveyor21IO.xCWPresent:=X37;
Y137:=H2200Conveyor21IO.xMotorCW;
H2200Conveyor21IO.iDeviceID:=2221;

H2200Conveyor22(ConveyorMotor:=H2200Conveyor22IO);
H2200Conveyor22IO.xForward:=M73;
H2200Conveyor22IO.xCWPresent:=X38;
Y138:=H2200Conveyor22IO.xMotorCW;
H2200Conveyor22IO.xNegLimit:=X15;
M118:=H2200Conveyor22IO.xOverWidthAlarm;
M119:=H2200Conveyor22IO.xLimitAlarrm;
H2200Conveyor22IO.iDeviceID:=2222;

H1000Conveyor11(ConveyorMotor:=H1000Conveyor11IO);
H1000Conveyor11IO.xForward:=M75;
H1000Conveyor11IO.xCWPresent:=X3A;
Y13A:=H1000Conveyor11IO.xMotorCW;
H1000Conveyor11IO.iDeviceID:=1011;

H1000Conveyor12(ConveyorMotor:=H1000Conveyor12IO);
H1000Conveyor12IO.xForward:=M76;
H1000Conveyor12IO.xCWPresent:=X3B;
Y13B:=H1000Conveyor12IO.xMotorCW;
H1000Conveyor12IO.iDeviceID:=1012;

H1000Conveyor13(ConveyorMotor:=H1000Conveyor13IO);
H1000Conveyor13IO.xForward:=M77;
H1000Conveyor13IO.xCWPresent:=X3C;
Y13C:=H1000Conveyor13IO.xMotorCW;
H1000Conveyor13IO.iDeviceID:=1013;

H1000Conveyor14(ConveyorMotor:=H1000Conveyor14IO);
H1000Conveyor14IO.xForward:=M78;
H1000Conveyor14IO.xCWPresent:=X3D;
Y13D:=H1000Conveyor14IO.xMotorCW;
H1000Conveyor14IO.iDeviceID:=1014;

H1000Conveyor15(ConveyorMotor:=H1000Conveyor15IO);
H1000Conveyor15IO.xForward:=M79;
H1000Conveyor15IO.xCWPresent:=X3E;
Y13E:=H1000Conveyor15IO.xMotorCW;
H1000Conveyor15IO.iDeviceID:=1015;

H1000Rotor2(ShuttleCarInOut:=H1000Rotor2IO);
ShuttleCarCurrentPosition( X9F OR X9E ,X9F ,X9E, FALSE, H1000Rotor2IO.iCurrentPos );
H1000Rotor2IO.xReady:=TRUE;
H1000Rotor2IO.xForward:=M93;
H1000Rotor2IO.xBackward:=M94;
H1000Rotor2IO.xPosLimit:=XB0;
H1000Rotor2IO.xNegLimit:=XB1;
Y1BC:=H1000Rotor2IO.xCW;
Y1BD:=H1000Rotor2IO.xCCW;
Y12A:=H1000Rotor2IO.xBrake;

H1000Rotor2Cylinder(ShuttleCarInOut:=H1000Rotor2CylinderIO);
ShuttleCarCurrentPosition( XA0 OR XA1 ,XA1 ,XA0, FALSE, H1000Rotor2CylinderIO.iCurrentPos );
H1000Rotor2CylinderIO.xReady:=TRUE;
H1000Rotor2CylinderIO.xForward:=M87;
H1000Rotor2CylinderIO.xBackward:=M88;
H1000Rotor2CylinderIO.xPosLimit:=TRUE;
H1000Rotor2CylinderIO.xNegLimit:=TRUE;
Y1A1:=H1000Rotor2CylinderIO.xCW;
Y1A0:=H1000Rotor2CylinderIO.xCCW;

H1000Conveyor16(ConveyorMotor:=H1000Conveyor16IO);
H1000Conveyor16IO.xForward:=M80;
H1000Conveyor16IO.xCWPresent:=X3F OR XC8;
Y13F:=H1000Conveyor16IO.xMotorCW;
H1000Conveyor16IO.iDeviceID:=1016;

H1000Rotor1(ShuttleCarInOut:=H1000Rotor1IO);
ShuttleCarCurrentPosition( X9A OR X9B ,X9A ,X9B, FALSE, H1000Rotor1IO.iCurrentPos );
H1000Rotor1IO.xReady:=TRUE;
H1000Rotor1IO.xForward:=M83;
H1000Rotor1IO.xBackward:=M84;
H1000Rotor1IO.xPosLimit:=X99;
H1000Rotor1IO.xNegLimit:=X98;
Y104:=H1000Rotor1IO.xCW;
Y105:=H1000Rotor1IO.xCCW;
Y129:=H1000Rotor1IO.xBrake;

H1000Rotor1Cylinder(ShuttleCarInOut:=H1000Rotor1CylinderIO);
ShuttleCarCurrentPosition( X9D OR X9C ,X9D ,X9C, FALSE, H1000Rotor1CylinderIO.iCurrentPos );
H1000Rotor1CylinderIO.xReady:=TRUE;
H1000Rotor1CylinderIO.xForward:=M85;
H1000Rotor1CylinderIO.xBackward:=M86;
H1000Rotor1CylinderIO.xPosLimit:=TRUE;
H1000Rotor1CylinderIO.xNegLimit:=TRUE;
Y19C:=H1000Rotor1CylinderIO.xCW;
Y19B:=H1000Rotor1CylinderIO.xCCW;

H1000Conveyor19(ConveyorMotor:=H1000Conveyor19IO);
H1000Conveyor19IO.xForward:=M81;
(*H1000Conveyor19IO.xCWPresent:=NOT X42;*)
H1000Conveyor19IO.xCWPresent:=XCE;
Y142:=H1000Conveyor19IO.xMotorCW;
H1000Conveyor19IO.xPosLimit:= X42;
(*H1000Conveyor19IO.xPosLimit:=1;*)
H1000Conveyor19IO.iDeviceID:=1019;
H1000Conveyor19IO.tLoadDelay:=T#200ms;
M138:=h1000Conveyor19IO.xLimitAlarrm;

H1000Conveyor20(ConveyorMotor:=H1000Conveyor20IO);
H1000Conveyor20IO.xForward:=M82;
H1000Conveyor20IO.xCWPresent:=X43;
Y143:=H1000Conveyor20IO.xMotorCW;
H1000Conveyor20IO.iDeviceID:=1020;

H850Conveyor1Trans(ConveyorMotor:=H850Conveyor1IOTrans);
H850Conveyor1IOTrans.xForward:=M120;
H850Conveyor1IOTrans.xCWPresent:=XA3;
Y1A3:=H850Conveyor1IOTrans.xMotorCW;
H850Conveyor1IOTrans.iDeviceID:=801;

H850Conveyor2Trans(ConveyorMotor:=H850Conveyor2IOTrans);
H850Conveyor2IOTrans.xForward:=M121;
H850Conveyor2IOTrans.xCWPresent:=XA4;
Y1A4:=H850Conveyor2IOTrans.xMotorCW;
H850Conveyor2IOTrans.iDeviceID:=802;

H850Conveyor3Trans(ConveyorMotor:=H850Conveyor3IOTrans);
H850Conveyor3IOTrans.xForward:=M122;
H850Conveyor3IOTrans.xCWPresent:=XA5;
Y1A5:=H850Conveyor3IOTrans.xMotorCW;
H850Conveyor3IOTrans.iDeviceID:=803;

H850Conveyor4Trans(ConveyorMotor:=H850Conveyor4IOTrans);
H850Conveyor4IOTrans.xForward:=M123;
H850Conveyor4IOTrans.xCWPresent:=XA6;
Y1A6:=H850Conveyor4IOTrans.xMotorCW;
H850Conveyor4IOTrans.iDeviceID:=804;

H850Conveyor5Trans(ConveyorMotor:=H850Conveyor5IOTrans);
H850Conveyor5IOTrans.xForward:=M124;
H850Conveyor5IOTrans.xCWPresent:=XA7;
Y1A7:=H850Conveyor5IOTrans.xMotorCW;
H850Conveyor5IOTrans.iDeviceID:=805;

H850Conveyor6Trans(ConveyorMotor:=H850Conveyor6IOTrans);
H850Conveyor6IOTrans.xForward:=M125;
H850Conveyor6IOTrans.xCWPresent:=XA8;
Y1A8:=H850Conveyor6IOTrans.xMotorCW;
H850Conveyor6IOTrans.iDeviceID:=806;

H850Conveyor7Trans(ConveyorMotor:=H850Conveyor7IOTrans);
H850Conveyor7IOTrans.xForward:=M126;
H850Conveyor7IOTrans.xCWPresent:=XA9;
Y1A9:=H850Conveyor7IOTrans.xMotorCW;
H850Conveyor7IOTrans.iDeviceID:=807;

H850Conveyor8Trans(ConveyorMotor:=H850Conveyor8IOTrans);
H850Conveyor8IOTrans.xForward:=M127;
H850Conveyor8IOTrans.xCWPresent:=XBA;
Y1AA:=H850Conveyor8IOTrans.xMotorCW;
H850Conveyor8IOTrans.iDeviceID:=808;

H380EmptyABumperBar( AccumulateConveyorIO:= H380EmptyABumperBarIO);
H380EmptyABumperBarIO.xBarCylinderButton:=M68;
H380EmptyABumperBarIO.xTransportMotorCWButton:=M89;
H380EmptyABumperBarIO.xTransportMotorCCWButton:=M90;
(*H380EmptyABumperBarIO.xPresentSwitch:=X48;*)
H380EmptyABumperBarIO.xPresentSwitchEntry:=X49;
Y148:=H380EmptyABumperBarIO.xBarCylinderSecondary OR M154;
Y149:=H380EmptyABumperBarIO.xBarCylinder OR M155;
Y15E:=H380EmptyABumperBarIO.xTransportMotorCW OR M156 ;(*往左为正转，下料方向为正*)
Y15D:=H380EmptyABumperBarIO.xTransportMotorCCW OR M157;
H380EmptyABumperBarIO.xTwoWay:=1;
H380EmptyABumperBarIO.tLoadDelay:=t#3S;
H380EmptyABumperBarIO.iDeviceID:=901;

H380EmptyARotorConveyor(ConveyorMotor:=H380EmptyARotorConveyorIO);
H380EmptyARotorConveyorIO.xCWPresent:=X7F;
H380EmptyARotorConveyorIO.xCCWPresent:=X7F;
H380EmptyARotorConveyorIO.tLoadDelay:=T#3S;
H380EmptyARotorConveyorIO.iDeviceID:=901;

H380EmptyALifter(ShuttleCarInOut:=H380EmptyALifterIO);(**升降**)
ShuttleCarCurrentPosition(  XC2 OR XC3 ,XC2 ,XC3,FALSE, H380EmptyALifterIO.iCurrentPos );
H380EmptyALifterIO.xReady:=TRUE;
H380EmptyALifterIO.xForward:=M26;
H380EmptyALifterIO.xBackward:=M27;
H380EmptyALifterIO.xPosLimit:=TRUE;
H380EmptyALifterIO.xNegLimit:=TRUE;
Y1D9:=H380EmptyALifterIO.xCW;
Y1DA:=H380EmptyALifterIO.xCCW;

H380EmptyARotor(ShuttleCarInOut:=H380EmptyARotorIO);(**旋转**)
ShuttleCarCurrentPosition( XC4 OR XC5 ,XC4 ,XC5, FALSE, H380EmptyARotorIO.iCurrentPos );
H380EmptyARotorIO.xReady:=TRUE;
H380EmptyARotorIO.xForward:=M28;
H380EmptyARotorIO.xBackward:=M29;
H380EmptyARotorIO.xPosLimit:=TRUE;
H380EmptyARotorIO.xNegLimit:=TRUE;
Y1D7:=H380EmptyARotorIO.xCW;(*逆时针为正*)
Y1D8:=H380EmptyARotorIO.xCCW;
H380EmptyARotorIO.xCylinder:=1;


H380EmptyBBumperBar(AccumulateConveyorIO:= H380EmptyBBumperBarIO);
H380EmptyBBumperBarIO.xBarCylinderButton:=M69;
H380EmptyBBumperBarIO.xTransportMotorCWButton:=M91;
H380EmptyBBumperBarIO.xTransportMotorCCWButton:=M92;
(*H380EmptyBBumperBarIO.xPresentSwitch:=X4A;*)
H380EmptyBBumperBarIO.xPresentSwitchEntry:=X4B;
Y14B:=H380EmptyBBumperBarIO.xBarCylinder OR M150;
Y1DD:=H380EmptyBBumperBarIO.xBarCylinderSecondary OR M151;
Y160:=H380EmptyBBumperBarIO.xTransportMotorCW OR M152;(*往右为正转*)
Y15F:=H380EmptyBBumperBarIO.xTransportMotorCCW OR M153;
H380EmptyBBumperBarIO.xTwoWay:=1;
H380EmptyBBumperBarIO.tLoadDelay:=t#3S;
H380EmptyBBumperBarIO.iDeviceID:=902;

H380EmptyBRotorConveyor(ConveyorMotor:=H380EmptyBRotorConveyorIO);
H380EmptyBRotorConveyorIO.xCWPresent:=XC1;
H380EmptyBRotorConveyorIO.xCCWPresent:=XC1;
H380EmptyBRotorConveyorIO.tLoadDelay:=T#3S;
H380EmptyBRotorConveyorIO.iDeviceID:=902;

H380EmptyBLifter(ShuttleCarInOut:=H380EmptyBLifterIO);(**升降**)
ShuttleCarCurrentPosition( XBC OR XBB ,XBC ,XBB, FALSE, H380EmptyBLifterIO.iCurrentPos );
H380EmptyBLifterIO.xReady:=TRUE;
H380EmptyBLifterIO.xForward:=M98;
H380EmptyBLifterIO.xBackward:=M99;
H380EmptyBLifterIO.xPosLimit:=TRUE;
H380EmptyBLifterIO.xNegLimit:=TRUE;
Y1D1:=H380EmptyBLifterIO.xCW;
Y1D2:=H380EmptyBLifterIO.xCCW;

H380EmptyBRotor(ShuttleCarInOut:=H380EmptyBRotorIO);(**旋转**)
ShuttleCarCurrentPosition( XBF OR XBD ,XBD ,XBF, FALSE, H380EmptyBRotorIO.iCurrentPos );
H380EmptyBRotorIO.xReady:=TRUE;
H380EmptyBRotorIO.xForward:=M100;
H380EmptyBRotorIO.xBackward:=M101;
H380EmptyBRotorIO.xPosLimit:=TRUE;
H380EmptyBRotorIO.xNegLimit:=TRUE;
Y1D3:=H380EmptyBRotorIO.xCW;(*逆时针为正*)
Y1D4:=H380EmptyBRotorIO.xCCW;
H380EmptyBRotorIO.xCylinder:=1;

(*自动状态*)
IF g_xAuto THEN
	(*上位机通讯扫码*)
(*	"化成RGV分流
4010"	2345	5	内衬型号	2345	"0：复位
1：读码失败
2：A筐内衬
3：B筐内衬"	3345	5	有板状态	3345	1：无板，2：有板*)
	IF H1000Conveyor19IO.xEmpty THEN
		D3345:=1;
	ELSE
		D3345:=2;
	END_IF;
   D225:=D2345;(*发送给RGV*)	
   (*D2345:=1;(*临时程序*)	
(*"提升机5二封满筐分流
4011"	2350	5	内衬型号	2350	"0：复位
1：读码失败
2：A筐内衬
3：B筐内衬"	3350	5	有板状态	3350	1：无板，2：有板*)
   IF h850Conveyor2IO.xEmpty THEN
   	D3350:=1;
   ELSE
   	D3350:=2;
   END_IF;
   D245:=D2350;
 (*"提升机4空框回流解绑
4012"	2355	5	步号解绑	2355	"0：复位
1：读码失败
2：A筐内衬
3：B筐内衬"	3355	5	有板状态	3355	1：无板，2：有板*)
  IF H850Conveyor1IO.xEmpty AND Lifter4IO.iCurrentPos=1THEN (*增加提升机到1号位置，才给扫码枪发信号*)
  	D3355:=1;
  ELSE
  	D3355:=2;
  END_IF;
 (* m_xDebindCode:=D2355=2;*)
	(********3000线体满框去二封************)
	D201.0:=H3000Conveyor11IO.xEmpty;
	H3000Conveyor11IO.xLoad:=D401.0;
	H3000Conveyor11IO.xUnload:=H3000Conveyor12IO.xEmpty;
	H3000Conveyor12IO.xLoad:=H3000Conveyor11IO.xNextRun;
	H3000Conveyor12IO.xUnload:=H3000Conveyor13IO.xEmpty;
	H3000Conveyor13IO.xLoad:=H3000Conveyor12IO.xNextRun;	
	H3000Conveyor13IO.xUnload:=H3000Conveyor14IO.xEmpty;
	H3000Conveyor14IO.xLoad:=H3000Conveyor13IO.xNextRun;
	H3000Conveyor14IO.xUnload:=H3000Conveyor15IO.xEmpty;
	H3000Conveyor15IO.xLoad:=H3000Conveyor14IO.xNextRun;
	H3000Conveyor15IO.xUnload:=H3000Conveyor16IO.xEmpty;
	H3000Conveyor16IO.xLoad:=H3000Conveyor15IO.xNextRun;
	H3000Conveyor16IO.xUnload:=H3000Conveyor17IO.xEmpty;
	H3000Conveyor17IO.xLoad:=H3000Conveyor16IO.xNextRun;
	H3000Conveyor17IO.xUnload:=H3000Conveyor18IO.xEmpty;
	H3000Conveyor18IO.xLoad:=H3000Conveyor17IO.xNextRun;	
	H3000Conveyor18IO.xUnload:=H3000Conveyor19IO.xEmpty;
	H3000Conveyor19IO.xLoad:=H3000Conveyor18IO.xNextRun;	
	H3000Conveyor19IO.xUnload:=H3000Conveyor20IO.xEmpty;
	H3000Conveyor20IO.xLoad:=H3000Conveyor19IO.xNextRun;
	H3000Conveyor20IO.xUnload:=H3000Conveyor21IO.xEmpty;
	H3000Conveyor21IO.xLoad:=H3000Conveyor20IO.xNextRun;
	H3000Conveyor21IO.xUnload:=H3000Conveyor22IO.xEmpty;
	H3000Conveyor22IO.xLoad:=H3000Conveyor21IO.xNextRun;
		(********3000线体满框去二封提升机************)
	IF Lifter5IO.iCurrentPos=2 AND X6F  THEN
		H3000Conveyor22IO.xUnload:=Conveyor5IO.xEmpty;
	ELSE
		H3000Conveyor22IO.xUnload:=0;		
	END_IF;
	conveyor5Io.xLoad:=H3000Conveyor22Io.xNextRun;
	IF Conveyor5IO.xEmpty  THEN
		Lifter5IO.xMDIExe:=1;
		Lifter5IO.iDestinationPos:=2;
	END_IF;
	IF Conveyor5IO.xEmpty=0 THEN
		Lifter5io.xMDIExe:=1;
		Lifter5IO.iDestinationPos:=1;
	END_IF;
	IF ldp(TRUE,Conveyor5IO.xEmpty=0) THEN
		D10:=D10+1;
	END_IF;
	IF  M74 THEN
		D10:=0;
	END_IF;
IF  Lifter5IO.iCurrentPos=1 AND X6E  THEN
	Conveyor5IO.xUnload:=H850Conveyor2IO.xEmpty;
ELSE
	Conveyor5IO.xUnload:=0;
END_IF;
	H850Conveyor2IO.xLoad:=Conveyor5IO.xNextRun;
	H850Conveyor2IO.xPutInto:=M881;(*临时程序*)
   (********3000线体满框去二封AGV接料************)
   (*发送*)
   D242.0:=QuarPackageRGV.xMdiExe;
   D242.1:=H850Conveyor1IOTrans.xEmpty;
   D242.2:=H850Conveyor2IOTrans.xEmpty;
   D242.3:=H850Conveyor3IOTrans.xEmpty;
   D242.4:=H850Conveyor4IOTrans.xEmpty;
   D242.5:=H850Conveyor5IOTrans.xEmpty;
   D242.6:=H850Conveyor6IOTrans.xEmpty;
   D242.7:=H850Conveyor7IOTrans.xEmpty;
   D242.8:=H850Conveyor8IOTrans.xEmpty;
   D242.9:=H850Conveyor1IO.xEmpty;
   D242.A:=H850Conveyor2IO.xEmpty;
   D242.B:=QuarPackageRGV.xAuto;
   D241:=QuarPackageRGV.iDestinationPos;
   D243.0:=QuarPackageRGV.xRemoteReset;
   D243.1:=H850Conveyor1IOTrans.xNextRun;
   D243.2:=H850Conveyor2IOTrans.xNextRun;
   D243.3:=H850Conveyor3IOTrans.xNextRun;
   D243.4:=H850Conveyor4IOTrans.xNextRun;
   D243.5:=H850Conveyor5IOTrans.xNextRun;
   D243.6:=H850Conveyor6IOTrans.xNextRun;
   D243.7:=H850Conveyor7IOTrans.xNextRun;
   D243.8:=H850Conveyor8IOTrans.xNextRun;
   D243.9:=H850Conveyor1IO.xNextRun;
   D243.A:=H850Conveyor2IO.xNextRun;
   QuarPackageRGV.xRemoteReset:=M137;
   QuarPackageRGV.xAuto:=M136;
    (*接收*)
   QuarPackageRGV.xMdiDone:=D432.0;
   H850Conveyor1IOTrans.xLoad:= D432.1;
   (*H850Conveyor2IOTrans.xLoad:= D432.2;  *)
   H850Conveyor3IOTrans.xLoad:= D432.3;
   (*H850Conveyor4IOTrans.xLoad:= D432.4; *)
   H850Conveyor5IOTrans.xLoad:= D432.5;
  (* H850Conveyor6IOTrans.xLoad:= D432.6; *)
   H850Conveyor7IOTrans.xLoad:= D432.7;
  (* H850Conveyor8IOTrans.xLoad:= D432.8;*)
   H850Conveyor1IO.xLoad:= D432.9 OR M880;
   (*H850Conveyor2IO.xLoad:= D432.A;*)
   QuarPackageRGV.iCurrentPostion:=D431;
   QuarPackageRGV.xCollisionAlarm:=D433.0;
 (*  H850Conveyor1IOTrans.xUnload:= D433.1;*)
   H850Conveyor2IOTrans.xUnload:= D433.2;
 (*  H850Conveyor3IOTrans.xUnload:= D433.3;*)
   H850Conveyor4IOTrans.xUnload:= D433.4;
 (*  H850Conveyor5IOTrans.xUnload:= D433.5;*)
   H850Conveyor6IOTrans.xUnload:= D433.6;
  (* H850Conveyor7IOTrans.xUnload:= D433.7;*)
   H850Conveyor8IOTrans.xUnload:= D433.8;
   (*H850Conveyor1IO.xUnload:= D433.9;*)
   H850Conveyor2IO.xUnload:= D433.A ;
	(*****************************二封1号机机对接信号******************************)
	QuarPackage1Stub.xUnloadRequestAkn:=XAE;
	QuarPackage1Stub.xLoadRequest:=XB2;
	Y1B0:=QuarPackage1Stub.xUnloadRequest;
	Y1B1:=QuarPackage1Stub.xLoadRequestAkn;
	
	H850Conveyor2IOTrans.xLoad:=QuarPackage1Stub.xLoadRequest;
	QuarPackage1Stub.xLoadRequestAkn:=H850Conveyor2IOTrans.xEmpty;
	H850Conveyor1IOTrans.xUnload:=QuarPackage1Stub.xUnloadRequestAkn;
	QuarPackage1Stub.xUnloadRequest:=NOT H850Conveyor1IOTrans.xEmpty;
		(*自动复位程序*)
	H850Conveyor1IOTrans.xPutInto:=NOT H850Conveyor1IOTrans.xBusy AND SM412;
	H850Conveyor2IOTrans.xPutInto:=NOT H850Conveyor2IOTrans.xBusy AND SM412;
	(*****************************二封2号机机对接信号******************************)	
	QuarPackage2Stub.xUnloadRequestAkn:=XB3;
	QuarPackage2Stub.xLoadRequest:=XB5;
	Y1B3:=QuarPackage2Stub.xUnloadRequest;
	Y1B4:=QuarPackage2Stub.xLoadRequestAkn;
	
	H850Conveyor4IOTrans.xLoad:=QuarPackage2Stub.xLoadRequest;
	QuarPackage2Stub.xLoadRequestAkn:=H850Conveyor4IOTrans.xEmpty;
	H850Conveyor3IOTrans.xUnload:=QuarPackage2Stub.xUnloadRequestAkn;
	QuarPackage2Stub.xUnloadRequest:=NOT H850Conveyor3IOTrans.xEmpty;
	
	(*自动复位程序*)
	H850Conveyor4IOTrans.xPutInto:=NOT H850Conveyor4IOTrans.xBusy AND SM412;
	H850Conveyor3IOTrans.xPutInto:=NOT H850Conveyor3IOTrans.xBusy AND SM412;
	(*****************************二封3号机机对接信号******************************)	
	QuarPackage3Stub.xUnloadRequestAkn:=XB6;
	QuarPackage3Stub.xLoadRequest:=XB8;
	Y1B6:=QuarPackage3Stub.xUnloadRequest;
	Y1B7:=QuarPackage3Stub.xLoadRequestAkn;
	
	H850Conveyor6IOTrans.xLoad:=QuarPackage3Stub.xLoadRequest;
	QuarPackage3Stub.xLoadRequestAkn:=H850Conveyor6IOTrans.xEmpty;
	H850Conveyor5IOTrans.xUnload:=QuarPackage3Stub.xUnloadRequestAkn;
	QuarPackage3Stub.xUnloadRequest:=NOT H850Conveyor5IOTrans.xEmpty;
	
	H850Conveyor6IOTrans.xPutInto:=NOT H850Conveyor6IOTrans.xBusy AND SM412;
	H850Conveyor5IOTrans.xPutInto:=NOT H850Conveyor5IOTrans.xBusy AND SM412;
	(*****************************二封4号机机对接信号******************************)
	QuarPackage4Stub.xUnloadRequestAkn:=XB9;
	QuarPackage4Stub.xLoadRequest:=XAB;
	Y1B9:=QuarPackage4Stub.xUnloadRequest;
	Y1BA:=QuarPackage4Stub.xLoadRequestAkn;
		
	H850Conveyor8IOTrans.xLoad:=QuarPackage4Stub.xLoadRequest;
	QuarPackage4Stub.xLoadRequestAkn:=H850Conveyor8IOTrans.xEmpty;
	H850Conveyor7IOTrans.xUnload:=QuarPackage4Stub.xUnloadRequestAkn;
	QuarPackage4Stub.xUnloadRequest:=NOT H850Conveyor7IOTrans.xEmpty;
	
	H850Conveyor8IOTrans.xPutInto:=NOT H850Conveyor8IOTrans.xBusy AND SM412;
	H850Conveyor7IOTrans.xPutInto:=NOT H850Conveyor7IOTrans.xBusy AND SM412;
	(******************************二封空框回流框型任务分配******************************)
	
	
	
	
	(*****************************二封前端RGV对接信号******************************)	  
      (*5号提升机接料位置满料*)
     IF M149 THEN
    QuarPackageRGV.xMdiExe:=1;
   	QuarPackageRGV.iDestinationPos:=6;
     END_IF;    
         (*4号提升机接料位置空框*) 	
    IF M135 THEN
   	QuarPackageRGV.xMdiExe:=1;
   	QuarPackageRGV.iDestinationPos:=5;
    END_IF;  
       (*1号上料*)
   IF M131 THEN
   	QuarPackageRGV.xMdiExe:=1;
   	QuarPackageRGV.iDestinationPos:=4;
   END_IF;
       (*2号上料*)
     IF M132 THEN
   	QuarPackageRGV.xMdiExe:=1;
   	QuarPackageRGV.iDestinationPos:=3;
     END_IF; 
         (*3号上料*)
    IF M133 THEN
   		QuarPackageRGV.xMdiExe:=1;
   		QuarPackageRGV.iDestinationPos:=2;
    END_IF;
          (*4号上料*)
   IF M134 THEN
   	QuarPackageRGV.xMdiExe:=1;
   	QuarPackageRGV.iDestinationPos:=1;
   END_IF;   	
   
	(********二封空框返回************)
    IF Conveyor4IO.xEmpty THEN
    	Lifter4Io.xMDIExe:=1;
    	Lifter4Io.iDestinationPos:=1;
    END_IF;
    IF Lifter4IO.iCurrentPos=1 AND X64   THEN
    	H850Conveyor1IO.xUnload:=Conveyor4Io.xEmpty AND D2355>1 ;	(********扫码成功放行********)
    ELSE
    	H850Conveyor1IO.xUnload:=0;
    END_IF;
       Conveyor4IO.xLoad:=H850Conveyor1IO.xNextRun;
       IF Conveyor4IO.xEmpty =0 AND Lifter4IO.iCurrentPos=1  THEN
       	   Lifter4IO.xMDIExe:=1;
       	   Lifter4IO.iDestinationPos:=2;
       END_IF;
       IF Lifter4IO.iCurrentPos=2 AND  X65   THEN
       	  Conveyor4IO.xUnload:=H2200Conveyor1IO.xEmpty;
       ELSE
       	 Conveyor4IO.xUnload:=0;
       END_IF;
       H2200Conveyor1IO.xLoad:=conveyor4IO.xNextRun;
   (********穿梭小车接空框************)
    IF ShuttleCar1IO.iCurrentPos=1 AND (NOT X53 AND NOT X54 ) THEN
        H2200Conveyor1IO.xUnload:=ConveyorShuttleCarIO.xEmpty;
    ELSE
    	H2200Conveyor1IO.xUnload:=0;
       	END_IF;
       	ConveyorShuttleCarIO.xLoad:= H2200Conveyor1IO.xNextRun;
      IF ConveyorShuttleCarIO.xEmpty  OR  M12 THEN   (********M12 回原点************)
        ShuttleCar1IO.xMDIExe:=1;
       	ShuttleCar1IO.iDestinationPos:=1;
      END_IF;     	
      
      (*M882空框回流A框与B框选择，触摸屏上按钮*)
       IF ConveyorShuttleCarIO.xEmpty =0 AND D2355=2   THEN
       	ShuttleCar1IO.xMDIExe:=1;
       	ShuttleCar1IO.iDestinationPos:=2;
       END_IF;
        IF ConveyorShuttleCarIO.xEmpty =0 AND   D2355=3   THEN
       	ShuttleCar1IO.xMDIExe:=1;
       	ShuttleCar1IO.iDestinationPos:=3;
        END_IF;
            IF (ShuttleCar1IO.iCurrentPos=2 AND NOT X53 AND NOT X55) 
       	    	OR (ShuttleCar1IO.iCurrentPos=3 AND  NOT X54 AND NOT X55 )  THEN
       	    	m_tofShuttleCar1LeaveDelay(IN:=ConveyorShuttleCarIO.xCWPresent ,PT:= T#5s ,Q:= m_xShuttleCar1LeaveDelay ,ET:= m_tShuttleCar1LeaveDelay );
       		    ConveyorShuttleCarIO.xUnload:= m_xShuttleCar1LeaveDelay;(*下料时间*)
       	    ELSE
       	        ConveyorShuttleCarIO.xUnload:=0;
       	    END_IF;
        
      (*空框回流A框与B框选择，*)
      (* IF ConveyorShuttleCarIO.xEmpty =0 AND ((m_iRGVEmptyTask =1 AND NOT D210.1)
       																			OR  (m_iRGVEmptyTask = 2  AND NOT  D210.2)
       																			OR  (m_iRGVEmptyTask =3  AND NOT D210.3)
       																			OR ( m_iRGVEmptyTask = 4 AND NOT D210.4) OR M20 ) THEN
       	ShuttleCar1IO.xMDIExe:=1;
       	ShuttleCar1IO.iDestinationPos:=2;
       END_IF;
        IF ConveyorShuttleCarIO.xEmpty =0 AND (( m_iRGVEmptyTask =1 AND  D210.1) 
        									   									OR  (m_iRGVEmptyTask = 2 AND  D210.2 ) 
        																		OR  (m_iRGVEmptyTask =3 AND  D210.3)
        	 																	OR  (m_iRGVEmptyTask =4 AND  D210.4)  OR M21 )  THEN
       	ShuttleCar1IO.xMDIExe:=1;
       	ShuttleCar1IO.iDestinationPos:=3;
       END_IF;     *)	

     (*空框回流A框与B框任务栈*)	
  (*   M22:=ConveyorShuttleCarIO.xEmpty AND  (m_iRGVEmptyTask =1 OR  m_iRGVEmptyTask =3 OR  m_iRGVEmptyTask =4) AND ShuttleCar1IO.iCurrentPos=2;
     M23:=ConveyorShuttleCarIO.xEmpty AND  m_iRGVEmptyTask =2  AND ShuttleCar1IO.iCurrentPos=3;
     
     RGVEmptyTask(arrxCondition:= m_arrxRGVEmptyTaskCondition ,  xTaskComplete:= LDp(TRUE,M22)  OR LDP (TRUE,M23 ) OR M24,xReset:= M24);
     
     m_iRGVEmptyTask:= RGVEmptyTask.iPriority ;*)	

		(*满框任务分配  任务栈式分配   *)  
	(*m_arrxRGVEmptyTaskCondition[1]:=H850Conveyor2IOTrans.xUnload ;
	m_arrxRGVEmptyTaskCondition[2]:=H850Conveyor4IOTrans.xUnload  AND FALSE ;
	m_arrxRGVEmptyTaskCondition[3]:=H850Conveyor6IOTrans.xUnload  ;
	m_arrxRGVEmptyTaskCondition[4]:=H850Conveyor8IOTrans.xUnload ;*)	
     
    (********H2200满框去化成***********)  
    D201.1:=  H2200Conveyor13IO.xEmpty;
	H2200Conveyor13IO.xLoad:=D401.1;
	H2200Conveyor13IO.xUnload:=H2200Conveyor14IO.xEmpty;
	H2200Conveyor14IO.xLoad:=H2200Conveyor13IO.xNextRun;
	H2200Conveyor14IO.xUnload:=H2200Conveyor15IO.xEmpty;
	H2200Conveyor15IO.xLoad:=H2200Conveyor14IO.xNextRun;	
	H2200Conveyor15IO.xUnload:=H2200Conveyor16IO.xEmpty;
	H2200Conveyor16IO.xLoad:=H2200Conveyor15IO.xNextRun;	
	H2200Conveyor16IO.xUnload:=H2200Conveyor17IO.xEmpty;
	H2200Conveyor17IO.xLoad:=H2200Conveyor16IO.xNextRun;	
	H2200Conveyor17IO.xUnload:=H2200Conveyor18IO.xEmpty;
	H2200Conveyor18IO.xLoad:=H2200Conveyor17IO.xNextRun;	
	H2200Conveyor18IO.xUnload:=H2200Conveyor19IO.xEmpty;
	H2200Conveyor19IO.xLoad:=H2200Conveyor18IO.xNextRun;		
	H2200Conveyor19IO.xUnload:=H2200Conveyor20IO.xEmpty;
	H2200Conveyor20IO.xLoad:=H2200Conveyor19IO.xNextRun;		
	H2200Conveyor20IO.xUnload:=H2200Conveyor21IO.xEmpty;
	H2200Conveyor21IO.xLoad:=H2200Conveyor20IO.xNextRun;		
	H2200Conveyor21IO.xUnload:=H2200Conveyor22IO.xEmpty;
	H2200Conveyor22IO.xLoad:=H2200Conveyor21IO.xNextRun;		
    IF conveyor3IO.xEmpty THEN
    	Lifter3IO.xMDIExe:=1;
    	Lifter3IO.iDestinationPos:=2;
    END_IF;
    IF conveyor3Io.xEmpty=0 THEN
      	Lifter3IO.xMDIExe:=1;
    	Lifter3IO.iDestinationPos:=1;  	
    END_IF;
    IF Lifter3IO.iCurrentPos=2 AND X5B THEN
    	H2200Conveyor22io.xUnload:= Conveyor3io.xEmpty;
    ELSE
    	H2200Conveyor22io.xUnload:=0;
    END_IF;
    Conveyor3IO.xLoad:=H2200Conveyor22io.xNextRun;
    IF Lifter3IO.iCurrentPos=1 AND X5A THEN
    	 Conveyor3IO.xUnload:=H1000Conveyor20IO.xEmpty;
    ELSE
    	 Conveyor3IO.xUnload:=0;
    END_IF;
    	H1000Conveyor20IO.xLoad:=Conveyor3IO.xNextRun;
    	H1000Conveyor20IO.xUnload:=H1000Conveyor19IO.xEmpty AND NOT h1000Conveyor19IO.xLimitAlarrm;
    	        IF ldp(TRUE,  H1000Conveyor20IO.xEmpty) THEN
    		D20:=D20+1;
    	END_IF;
    	(*清零程序*)
    	IF M97 THEN
    		D20:=0;
    	END_IF;
       H1000Conveyor19IO.xLoad:=H1000Conveyor20IO.xNextRun;
      H1000Conveyor19IO.xPutInto:=XD7;               
       (*化成RGV接料程序*)
       (*F线对接信号*)
       Chem1Stub.xLoadRequest:=X80;(*满框上料*)
       Chem1Stub.xUnloadRequest:=X81;(*空框下料*)
       Chem2Stub.xLoadRequest:=X82;(*空框上料*)
       Chem2Stub.xUnloadRequest:=X83;(*满框下料*)
       
       Y180:=Chem1Stub.xLoadRequestAkn;(*满框上料完成*)
       Y181:=Chem1Stub.xUnloadRequestAkn;(*空框下料完成*)
       Y182:=Chem2Stub.xLoadRequestAkn;(*空框上料完成*)
       Y183:=Chem2Stub.xUnloadRequestAkn; (*满框下料完成*)    
              (*E线对接信号*)
       Chem3Stub.xLoadRequest:=X84;(*满框上料*)
       Chem3Stub.xUnloadRequest:=X85;(*空框下料*)
       Chem4Stub.xLoadRequest:=X86;(*空框上料*)
       Chem4Stub.xUnloadRequest:=X87;(*满框下料*)
       
       Y184:=Chem3Stub.xLoadRequestAkn;(*满框上料完成*)
       Y185:=Chem3Stub.xUnloadRequestAkn;(*空框下料完成*)
       Y186:=Chem4Stub.xLoadRequestAkn;(*空框上料完成*)
       Y187:=Chem4Stub.xUnloadRequestAkn; (*满框下料完成*)   
              (*D线对接信号*)
       Chem5Stub.xLoadRequest:=X88;(*满框上料*)
       Chem5Stub.xUnloadRequest:=X89;(*空框下料*)
       Chem6Stub.xLoadRequest:=X8A;(*空框上料*)
       Chem6Stub.xUnloadRequest:=X8B;(*满框下料*)
       
       Y188:=Chem5Stub.xLoadRequestAkn;(*满框上料完成*)
       Y189:=Chem5Stub.xUnloadRequestAkn;(*空框下料完成*)
       Y18A:=Chem6Stub.xLoadRequestAkn;(*空框上料完成*)
       Y18B:=Chem6Stub.xUnloadRequestAkn; (*满框下料完成*)     
       (*C线对接信号*)
       Chem11Stub.xLoadRequest:=X8C;(*满框上料*)
       Chem11Stub.xUnloadRequest:=X8D;(*空框下料*)
       Chem12Stub.xLoadRequest:=X8E;(*空框上料*)
       Chem12Stub.xUnloadRequest:=X8F;(*满框下料*)
       
       Y18C:=Chem11Stub.xLoadRequestAkn;(*满框上料完成*)
       Y18D:=Chem11Stub.xUnloadRequestAkn;(*空框下料完成*)
       Y18E:=Chem12Stub.xLoadRequestAkn;(*空框上料完成*)
       Y18F:=Chem12Stub.xUnloadRequestAkn; (*满框下料完成*)  
              (*B线对接信号*)
       Chem9Stub.xLoadRequest:=X90;(*满框上料*)
       Chem9Stub.xUnloadRequest:=X91;(*空框下料*)
       Chem10Stub.xLoadRequest:=X92;(*空框上料*)
       Chem10Stub.xUnloadRequest:=X93;(*满框下料*)
       
       Y190:=Chem9Stub.xLoadRequestAkn;(*满框上料完成*)
       Y191:=Chem9Stub.xUnloadRequestAkn;(*空框下料完成*)
       Y192:=Chem10Stub.xLoadRequestAkn;(*空框上料完成*)
       Y193:=Chem10Stub.xUnloadRequestAkn; (*满框下料完成*)  
              (*A线对接信号*)
       Chem7Stub.xLoadRequest:=X94;(*满框上料*)
       Chem7Stub.xUnloadRequest:=X95;(*空框下料*)
       Chem8Stub.xLoadRequest:=X96;(*空框上料*)
       Chem8Stub.xUnloadRequest:=X97;(*满框下料*)
       
       Y194:=Chem7Stub.xLoadRequestAkn;(*满框上料完成*)
       Y195:=Chem7Stub.xUnloadRequestAkn;(*空框下料完成*)
       Y196:=Chem8Stub.xLoadRequestAkn;(*空框上料完成*)
       Y197:=Chem8Stub.xUnloadRequestAkn; (*满框下料完成*)  
	(*发送*)
   D221:=ChemRGV.iDestinationPos;	
   D222.0:=ChemRGV.xAuto; 	
   D222.1:=ChemRGV.xMdiExe;
   D222.2:=ChemRGV.xLoad1;
   D222.3:=ChemRGV.xUnload1;
   D222.4:=Chem1Stub.xLoadRequest;
   D222.5:=Chem2Stub.xLoadRequest;
   D222.6:=Chem3Stub.xLoadRequest;
   D222.7:=Chem4Stub.xLoadRequest;
   D222.8:=Chem5Stub.xLoadRequest;
   D222.9:=Chem6Stub.xLoadRequest;
   D222.A:=Chem7Stub.xLoadRequest;
   D222.B:=Chem8Stub.xLoadRequest;
   D222.C:=Chem9Stub.xLoadRequest;
   D222.D:=Chem10Stub.xLoadRequest;
   D222.E:=Chem11Stub.xLoadRequest;
   D222.F:=Chem12Stub.xLoadRequest;
     
   D223.0:=ChemRGV.xRemoteReset;
   D223.1:=Chem1Stub.xUnloadRequest;
   D223.2:=Chem2Stub.xUnloadRequest;
   D223.3:=Chem3Stub.xUnloadRequest;
   D223.4:=Chem4Stub.xUnloadRequest;  
   D223.5:=Chem5Stub.xUnloadRequest;
   D223.6:=Chem6Stub.xUnloadRequest;
   D223.7:=Chem7Stub.xUnloadRequest;
   D223.8:=Chem8Stub.xUnloadRequest;  
   D223.9:=Chem9Stub.xUnloadRequest; 
   D223.A:=Chem10Stub.xUnloadRequest;
   D223.B:=Chem11Stub.xUnloadRequest; 
   D223.C:=Chem12Stub.xUnloadRequest;  
   
   D224.0:=H1000Conveyor19IO.xEmpty;
   D224.1:=h1000Conveyor19IO.xNextRun;
   D224.2:=H1000Conveyor16IO.xEmpty; 
   D224.3:=H380EmptyARotorConveyorIO.xEmpty;
   D224.4:=H380EmptyABumperBarIO.xNextRun ;
   D224.5:=H380EmptyBRotorConveyorIO.xEmpty;
   D224.6:=H380EmptyBBumperBarIO.xNextRun;   
   
   ChemRGV.xRemoteReset:=M139;
   ChemRGV.xAuto:=M140 OR  XD5;
   (*接收*)
   ChemRGV.iCurrentPostion:=D421;
   Chem1Stub.xLoadRequestAkn:=D422.0;
   Chem2Stub.xLoadRequestAkn:=D422.1;
   Chem3Stub.xLoadRequestAkn:=D422.2;
  Chem4Stub.xLoadRequestAkn:=D422.3;
   Chem5Stub.xLoadRequestAkn:=D422.4;
   Chem6Stub.xLoadRequestAkn:= D422.5;
   Chem7Stub.xLoadRequestAkn:= D422.6; 
   Chem8Stub.xLoadRequestAkn:= D422.7; 
   Chem9Stub.xLoadRequestAkn:= D422.8;
    Chem10Stub.xLoadRequestAkn:= D422.9;
   Chem11Stub.xLoadRequestAkn:= D422.A; 
  Chem12Stub.xLoadRequestAkn:= D422.B; 

   ChemRGV.xCollisionAlarm:=D423.0;
   Chem1Stub.xUnloadRequestAkn:=D423.1;	
    Chem2Stub.xUnloadRequestAkn:=D423.2;
    Chem3Stub.xUnloadRequestAkn:=D423.3;	
    Chem4Stub.xUnloadRequestAkn:=D423.4;
    Chem5Stub.xUnloadRequestAkn:=D423.5;
    Chem6Stub.xUnloadRequestAkn:=D423.6;
    Chem7Stub.xUnloadRequestAkn:=D423.7;
    Chem8Stub.xUnloadRequestAkn:=D423.8;
    Chem9Stub.xUnloadRequestAkn:=D423.9;
    Chem10Stub.xUnloadRequestAkn:=D423.A;
    Chem11Stub.xUnloadRequestAkn:=D423.B;
    Chem12Stub.xUnloadRequestAkn:=D423.C;
    m_xDirection:=NOT (D423.D OR M161) ;
    m_xLoadDirection:=NOT D423.E;
    m_xUnloadDirection:=NOT D423.F;
    
    (*化成下料段按钮盒*)(*按3秒钟后执行下料，确保安全*)
    m_tonXD8(IN:= XD8  ,PT:= T#3S ,Q:= m_xXD8 ,ET:= m_tXD8);
    IF  m_xXD8 THEN
    	m_xXD8Lock:=1;
    END_IF;
    IF NOT D424.0 THEN
    	m_xXD8Lock:=0;
    END_IF;
    H1000Conveyor19IO.xUnload:=D424.0    (*RGV信号*)
    														(*AND m_xXD8Lock  (*下料按钮按3秒*)
    														AND (NOT m_xLoadDirection (*不需要旋转直接放行**)
    																OR ( m_xLoadDirection AND m_xRotor1Done) (*需要旋转，转完放行*)
    																OR ChemRGV.xAuto  );(*半自动模式直接放行*)
    m_xRotor1Start:=D424.0 AND m_xLoadDirection AND NOT ChemRGV.xAuto ; (*有下料信号，但没有方向信号，需要旋转*) 	
 	H1000Conveyor16IO.xLoad:=D424.1;
 	m_xRotor2Start:=H1000Conveyor16IO.xEmpty=0 AND m_xUnloadDirection AND NOT ChemRGV.xAuto;
 	
 (*右空框回流*)
  	H380EmptyABumperBarIO.xLoad :=D424.2;
  	H380EmptyARotorConveyorIO.xLoad:=H380EmptyARotorConveyorIO.xEmpty AND(H380EmptyABumperBarIO.xLoad OR H380EmptyABumperBarIO.xNextRun) ;
    H380EmptyARotorConveyorIO.xloadCCW:=D424.2;
    m_xEmptyARotorStart:=NOT H380EmptyARotorConveyorIO.xEmpty AND m_xDirection;
    H380EmptyARotorConveyorIO.xUnload:=((NOT H380EmptyABumperBarIO.xLoadDone AND H380EmptyABumperBarIO.xTransportMotorCCW)
    																					OR  H380EmptyABumperBarIO.xUnload ) 
    																					AND(NOT m_xDirection OR ( m_xDirection AND m_xEmptyARotorDone));
       IF H380EmptyARotorConveyorIO.xload AND H380EmptyARotorConveyorIO.xMotorCCW THEN
  	 	Y1DC:=0;(*转台左右两个阻挡*)
  	 	Y17E:=1;
		ELSIF H380EmptyARotorConveyorIO.xload AND H380EmptyARotorConveyorIO.xMotorCW THEN
	   	Y1DC:=1;
   		Y17E:=0;
 		ELSIF H380EmptyARotorConveyorIO.xNextRun THEN	
 		Y1DC:=1;
   		Y17E:=1;
   		END_IF;	
	H380EmptyABumperBarIO.xUnload:=D424.3;
	
 	(*左边的空框回流*)
  	H380EmptyBBumperBarIO.xLoad :=D424.4 ;
  	H380EmptyBRotorConveyorIO.xLoad:=H380EmptyBRotorConveyorIO.xEmpty AND(H380EmptyBBumperBarIO.xLoad OR H380EmptyBBumperBarIO.xNextRun) ;
    H380EmptyBRotorConveyorIO.xloadCCW:=D424.4;
    m_xEmptyBRotorStart:=NOT H380EmptyBRotorConveyorIO.xEmpty AND m_xDirection;
    H380EmptyBRotorConveyorIO.xUnload:=((NOT H380EmptyBBumperBarIO.xLoadDone AND H380EmptyBBumperBarIO.xTransportMotorCCW)
    																					OR  H380EmptyBBumperBarIO.xUnload ) 
    																					AND(NOT m_xDirection OR ( m_xDirection AND m_xEmptyBRotorDone));
       IF H380EmptyBRotorConveyorIO.xload AND H380EmptyBRotorConveyorIO.xMotorCCW THEN
  	 	Y17D:=0;(*转台左右两个阻挡*)
  	 	Y1D6:=1;
		ELSIF H380EmptyBRotorConveyorIO.xload AND H380EmptyBRotorConveyorIO.xMotorCW THEN
	   	Y17D:=1;
   		Y1D6:=0;
 		ELSIF H380EmptyBRotorConveyorIO.xNextRun THEN	
 		Y17D:=1;
   		Y1D6:=1;
   		END_IF;	
 	H380EmptyBBumperBarIO.xUnload:=D424.5 OR M160;
 	
      (*去空框上下料位置*)
    IF M141 THEN
   	ChemRGV.xMdiExe:=1;
   	ChemRGV.iDestinationPos:=8;
    END_IF;   
       (*满框上下料位置*)
   IF M142 THEN
   	ChemRGV.xMdiExe:=1;
   	ChemRGV.iDestinationPos:=7;
   END_IF;
       (*1号华成机满框上料，空框下料*)
     IF M143 THEN
   	ChemRGV.xMdiExe:=1;
   	ChemRGV.iDestinationPos:=6;
     END_IF; 
       (*1号华成机满框下料，空框上料*)
    IF M144 THEN
   		ChemRGV.xMdiExe:=1;
   		ChemRGV.iDestinationPos:=5;
    END_IF;
       (*2号华成机满框上料，空框下料*)
   IF M145 THEN
   	ChemRGV.xMdiExe:=1;
   	ChemRGV.iDestinationPos:=4;
   END_IF;   
      (*2号华成机满框下料，空框上料*)        
      IF M146 THEN
   	ChemRGV.xMdiExe:=1;
   	ChemRGV.iDestinationPos:=3;
      END_IF;  
        (*3号华成机满框上料，空框下料*)
   IF M147 THEN
   	ChemRGV.xMdiExe:=1;
   	ChemRGV.iDestinationPos:=2;
   END_IF;   
      (*3号华成机满框下料，空框上料*)        
      IF M148 THEN
   	ChemRGV.xMdiExe:=1;
   	ChemRGV.iDestinationPos:=1;
      END_IF;      
          
        (*化成RGV满框出料程序*)
        H1000Conveyor16IO.xLoad:=XD0 ;(*----加了个按钮*)
        IF XD2 OR D424.7 THEN
        	m_xCheckDone:=1;
        END_IF;
        IF H1000Conveyor16IO.xEmpty THEN
        	m_xCheckDone:=0;
        END_IF;
         H1000Conveyor16IO.xPutInto:=LDF(TRUE,XD0) ;
       H1000Conveyor16IO.xUnload:=H1000Conveyor15IO.xEmpty AND m_xCheckDone  (*AND (NOT m_xRotor1Start  OR (m_xRotor1Start AND m_xRotor1Done))*);
       (*化成下料转台旋转*)
       CASE m_iH1000Rotor2Step OF
       0:
       IF LDF(TRUE, XD1 OR D424.6)  OR LDP(TRUE,m_xRotor2Start)  THEN  (*手动按钮*)
       		m_iH1000Rotor2Step:=1;
       END_IF;
       1:(*顶升*)
		H1000Rotor2CylinderIO.xMDIExe:=1;
		H1000Rotor2CylinderIO.iDestinationPos:=2;  
		IF  H1000Rotor2CylinderIO.iCurrentPos =2 THEN
			m_iH1000Rotor2Step:=2;
		END_IF;
		2:(*旋转*)
			IF H1000Rotor2IO.iCurrentPos =1 THEN
				m_iH1000Rotor2Step:=3;
			END_IF;
			IF H1000Rotor2IO.iCurrentPos =2 THEN
				m_iH1000Rotor2Step:=4;
			END_IF;
			3:
			H1000Rotor2IO.xMDIExe:=1;
			H1000Rotor2IO.iDestinationPos:=2;
			IF H1000Rotor2IO.iCurrentPos =2 THEN
				m_iH1000Rotor2Step:=5; 	
			END_IF;
			4:
			H1000Rotor2IO.xMDIExe:=1;
			H1000Rotor2IO.iDestinationPos:=1;	
			IF H1000Rotor2IO.iCurrentPos =1 THEN
				m_iH1000Rotor2Step:=5; 	
			END_IF;				
			5:(*下降*)
			H1000Rotor2CylinderIO.xMDIExe:=1;
			H1000Rotor2CylinderIO.iDestinationPos:=1; 
			m_xRotor2Done:=1;	
			IF  H1000Rotor2CylinderIO.iCurrentPos =1 THEN
					m_iH1000Rotor2Step:=0;	
			END_IF;      		
       END_CASE;
       IF H1000Conveyor19IO.xEmpty THEN(*转台为空复位旋转完成信号*)
       		m_xRotor1Done:=0;	
       	END_IF;
        (*化成上料转台旋转*)
       CASE m_iH1000Rotor1Step OF
       0:
       IF LDF(TRUE, XD6) OR LDP (TRUE,m_xRotor1Start) THEN
       		m_iH1000Rotor1Step:=1;
       END_IF;
       1:
		H1000Rotor1CylinderIO.xMDIExe:=1;
		H1000Rotor1CylinderIO.iDestinationPos:=2;  
		IF  H1000Rotor1CylinderIO.iCurrentPos =2 THEN
			m_iH1000Rotor1Step:=2;
		END_IF;
		2:
			IF H1000Rotor1IO.iCurrentPos =1 THEN
				m_iH1000Rotor1Step:=3;
			END_IF;
			IF H1000Rotor1IO.iCurrentPos =2 THEN
				m_iH1000Rotor1Step:=4;
			END_IF;
			3:
			H1000Rotor1IO.xMDIExe:=1;
			H1000Rotor1IO.iDestinationPos:=2;
			IF H1000Rotor1IO.iCurrentPos =2 THEN
				m_iH1000Rotor1Step:=5; 	
			END_IF;
			4:
			H1000Rotor1IO.xMDIExe:=1;
			H1000Rotor1IO.iDestinationPos:=1;	
			IF H1000Rotor1IO.iCurrentPos =1 THEN
				m_iH1000Rotor1Step:=5; 	
			END_IF;				
			5:
			H1000Rotor1CylinderIO.xMDIExe:=1;
			H1000Rotor1CylinderIO.iDestinationPos:=1; 
			m_xRotor1Done:=1;		
			IF  H1000Rotor1CylinderIO.iCurrentPos =1 THEN
					m_iH1000Rotor1Step:=0;	
			END_IF;      		
       END_CASE;
        IF H1000Conveyor16IO.xEmpty THEN(*转台为空复位旋转完成信号*)
       		m_xRotor2Done:=0;	
       		m_xRotor2Start:=0;
       	END_IF;			
      TON_ARotorStep5(IN:= m_iEmptyARotorStep=5 ,PT:= T#500MS ,Q:= m_xARotorStep5 ,ET:= m_tARotorStep5); 	
       TON_BRotorStep5(IN:=m_iEmptyBRotorStep=5 ,PT:= T#500MS ,Q:= m_xBRotorStep5 ,ET:=m_tBRotorStep5 );	
	CASE m_iEmptyBRotorStep OF
       0:
       IF LDP(TRUE,m_xEmptyBRotorStart)  THEN  (*手动按钮*)
       		m_iEmptyBRotorStep:=1;
       END_IF;
       1:(*顶升and夹紧*)
		H380EmptyBLifterIO.xMDIExe:=1;
		H380EmptyBLifterIO.iDestinationPos:=2;  
		IF  H380EmptyBLifterIO.iCurrentPos =2 THEN
			Y1D5:=1;
		END_IF;
		IF H380EmptyBLifterIO.iCurrentPos =2 AND XBE THEN
			m_iEmptyBRotorStep :=2;
		END_IF;	
		2:(*旋转*)
			IF H380EmptyBRotorIO.iCurrentPos =1 THEN
				m_iEmptyBRotorStep :=3;
			END_IF;
			IF H380EmptyBRotorIO.iCurrentPos =2 THEN
				m_iEmptyBRotorStep :=4;
			END_IF;
			3:
			H380EmptyBRotorIO.xMDIExe:=1;
			H380EmptyBRotorIO.iDestinationPos:=2;
			IF H380EmptyBRotorIO.iCurrentPos =2 THEN
				m_iEmptyBRotorStep :=5; 	
			END_IF;
			4:
			H380EmptyBRotorIO.xMDIExe:=1;
			H380EmptyBRotorIO.iDestinationPos:=1;	
			IF H380EmptyBRotorIO.iCurrentPos =1 THEN
				m_iEmptyBRotorStep :=5; 	
			END_IF;				
			5:(*下降*)
			IF m_xBRotorStep5 THEN
			Y1D5:=0;
			END_IF;
			IF XC0 THEN
			H380EmptyBLifterIO.xMDIExe:=1;
			H380EmptyBLifterIO.iDestinationPos:=1; 
			m_xEmptyBRotorDone:=1;	
			END_IF;
			IF  H380EmptyBLifterIO.iCurrentPos =1 THEN
					m_iEmptyBRotorStep :=0;	
			END_IF;      		
      END_CASE;
       IF H380EmptyBRotorConveyorIO.xEmpty THEN(*转台为空复位旋转完成信号*)
       		m_xEmptyBRotorDone:=0;	
       	END_IF;
      	
    CASE m_iEmptyARotorStep OF
       0:
       IF LDP(TRUE,m_xEmptyARotorStart)  THEN  (*手动按钮*)
       		m_iEmptyARotorStep:=1;
       END_IF;
       1:(*顶升and夹紧*)
		H380EmptyALifterIO.xMDIExe:=1;
		H380EmptyALifterIO.iDestinationPos:=2;  
		IF  H380EmptyALifterIO.iCurrentPos =2 THEN
			Y1DB:=1;
		END_IF;
		IF H380EmptyALifterIO.iCurrentPos =2 AND XC6 THEN
			m_iEmptyARotorStep :=2;
		END_IF;	
		2:(*旋转*)
			IF H380EmptyARotorIO.iCurrentPos =1 THEN
				m_iEmptyARotorStep :=3;
			END_IF;
			IF H380EmptyARotorIO.iCurrentPos =2 THEN
				m_iEmptyARotorStep :=4;
			END_IF;
			3:
			H380EmptyARotorIO.xMDIExe:=1;
			H380EmptyARotorIO.iDestinationPos:=2;
			IF H380EmptyARotorIO.iCurrentPos =2 THEN
				m_iEmptyARotorStep :=5; 	
			END_IF;
			4:
			H380EmptyARotorIO.xMDIExe:=1;
			H380EmptyARotorIO.iDestinationPos:=1;	
			IF H380EmptyARotorIO.iCurrentPos =1 THEN
				m_iEmptyARotorStep :=5; 	
			END_IF;				
			5:(*下降*)
			IF m_xARotorStep5 THEN
			Y1DB:=0;
			END_IF;
			IF XC7 THEN
			H380EmptyALifterIO.xMDIExe:=1;
			H380EmptyALifterIO.iDestinationPos:=1; 
			m_xEmptyARotorDone:=1;	
			END_IF;
			IF  H380EmptyALifterIO.iCurrentPos =1 THEN
					m_iEmptyARotorStep :=0;	
			END_IF;      		
    END_CASE;
       IF H380EmptyARotorConveyorIO.xEmpty THEN(*转台为空复位旋转完成信号*)
       		m_xEmptyARotorDone:=0;	
       	END_IF;
      	

      	
        IF ldp(TRUE,  H1000Conveyor15IO.xEmpty) THEN
    		D22:=D22+1;
    	END_IF;
    	(*清零程序*)
    	IF M96 THEN
    		D22:=0;
    	END_IF;
    	
    	
       H1000Conveyor15IO.xLoad:=H1000Conveyor16IO.xNextRun ;
        H1000Conveyor15IO.xUnload:=H1000Conveyor14IO.xEmpty;
       H1000Conveyor14IO.xLoad:=H1000Conveyor15IO.xNextRun;
            
          (***-------以下部分是RGV下料位置增加了个全检工位，m_xAllCheck信号为1，上料完毕就停下等待检查，检查完毕按下m_xAllCheckOver表示检查完毕，等下段空就下料，
          ----------------如果m_xAllCheck没信号，就直接等下段空就开始下料***)
        m_xAllCheck:=X41;
        m_xAllCheckOver:=X40;
                IF ldp(TRUE,m_xAllCheckOver) THEN
       	             m_xPassAllow:=1;
                END_IF;
                IF ldf(TRUE,H1000Conveyor13IO.xEmpty )  
                	OR( g_xResetSingle AND  H1000Conveyor14IO.iDeviceID=g_iDeviceIDSelect)
                   OR g_xReset  OR NOT m_xAllCheck THEN
                	m_xPassAllow:=0;
                END_IF;                     
         H1000Conveyor14IO.xUnload:=H1000Conveyor13IO.xEmpty AND ( m_xAllCheck AND m_xPassAllow OR NOT m_xAllCheck);
         (**---------------这里把那个putinto信号拿来复位超宽报警了，不知道有没有坏的影响***)
        IF ldp(TRUE,XD7)THEN
        	H1000Conveyor19IO.xOverWidthAlarm:=0;
        	END_IF;
         
       H1000Conveyor13IO.xLoad:=H1000Conveyor14IO.xNextRun; 
        H1000Conveyor13IO.xUnload:=H1000Conveyor12IO.xEmpty;
       H1000Conveyor12IO.xLoad:=H1000Conveyor13IO.xNextRun;
        H1000Conveyor13IO.xUnload:=H1000Conveyor12IO.xEmpty;
       H1000Conveyor12IO.xLoad:=H1000Conveyor13IO.xNextRun;
        H1000Conveyor12IO.xUnload:=H1000Conveyor11IO.xEmpty;
       H1000Conveyor11IO.xLoad:=H1000Conveyor12IO.xNextRun;      
      H1000Conveyor11IO.xUnload:=D401.2;(*接收给化成1号柜*线体10为空信号*)
      D201.2:=    H1000Conveyor11IO.xNextRun;(*发送给化成1号柜*线体10为开始旋转信号*)
END_IF;
 Y158:=M66 AND g_xEStop ;(*空框A返回倍速链*)
 Y15A:=M67 AND g_xEStop;(*空框B返回倍速链*)
 
 (*注液到化成空框A线*)
 (*H2200SudsecitonCylinderA3(BarCylinderIO:= H2200SudsecitonCylinderA3IO );(*空框回流分段阻挡气缸*)
(*H2200SudsecitonCylinderA3IO.xBarCylinderButton:=M212;
H2200SudsecitonCylinderA3IO.xPresentSwitch:=X36;
???:=H2200SudsecitonCylinderA3IO.xBarCylinder;*)(*******气缸还没装先屏蔽这段******)
 
 H2200SudsecitonCylinderA4(BarCylinderIO:= H2200SudsecitonCylinderA4IO );(*空框回流分段阻挡气缸*)
H2200SudsecitonCylinderA4IO.xBarCylinderButton:=M213;
H2200SudsecitonCylinderA4IO.xPresentSwitch:=X38;
Y174:=H2200SudsecitonCylinderA4IO.xBarCylinder;

H2200SudsecitonCylinderA5(BarCylinderIO:= H2200SudsecitonCylinderA5IO );(*空框回流分段阻挡气缸*)
H2200SudsecitonCylinderA5IO.xBarCylinderButton:=M214;
H2200SudsecitonCylinderA5IO.xPresentSwitch:=X3E;
Y171:=H2200SudsecitonCylinderA5IO.xBarCylinder;

(*m_tonSudsecitonCylinderA3Delay(IN:= NOT X5E AND NOT XC1,
											PT:=T#10s,
											Q:= H2200SudsecitonCylinderA3IO.xUnload,
											ET:=m_tCylinderA3DelayCurrentTime);
IF X5E THEN
	H2200SudsecitonCylinderA3IO.xUnload:=0;
	END_IF;
END_IF;*)             (*******气缸还没装先屏蔽这段******)

(*IF NOT X36 AND NOT X37 THEN*)
m_tonSudsecitonCylinderA4Delay(IN:= NOT X5E AND NOT XC1,
											PT:=T#10s,
											Q:= H2200SudsecitonCylinderA4IO.xUnload,
											ET:=m_tCylinderA4DelayCurrentTime);
IF X5E THEN
	(*ELSIF X36 THEN*)
	H2200SudsecitonCylinderA4IO.xUnload:=0;
END_IF;

m_tonSudsecitonCylinderA5Delay(IN:= NOT X38 AND NOT X39,
											PT:=T#10s,
											Q:= H2200SudsecitonCylinderA5IO.xUnload,
											ET:=m_tCylinderA5DelayCurrentTime);
IF X38 THEN
	H2200SudsecitonCylinderA5IO.xUnload:=0;
END_IF;

IF  X3E AND  X31 THEN
	BlockA:=1;
	ELSIF NOT X3E THEN
	BlockA:=0;
END_IF;

 (*注液到化成空框B线*)
 (*H2200SudsecitonCylinderB3(BarCylinderIO:= H2200SudsecitonCylinderB3IO );(*空框回流分段阻挡气缸*)
(*H2200SudsecitonCylinderB3IO.xBarCylinderButton:=M217;
H2200SudsecitonCylinderB3IO.xPresentSwitch:=X3A;
???:=H2200SudsecitonCylinderB3IO.xBarCylinder;*)(*******气缸还没装先屏蔽这段******)

H2200SudsecitonCylinderB4(BarCylinderIO:= H2200SudsecitonCylinderB4IO );(*空框回流分段阻挡气缸*)
H2200SudsecitonCylinderB4IO.xBarCylinderButton:=M218;
H2200SudsecitonCylinderB4IO.xPresentSwitch:=X3C;
Y172:=H2200SudsecitonCylinderB4IO.xBarCylinder;

H2200SudsecitonCylinderB5(BarCylinderIO:= H2200SudsecitonCylinderB5IO );(*空框回流分段阻挡气缸*)
H2200SudsecitonCylinderB5IO.xBarCylinderButton:=M219;
H2200SudsecitonCylinderB5IO.xPresentSwitch:=X40;
Y170:=H2200SudsecitonCylinderB5IO.xBarCylinder;

(*m_tonSudsecitonCylinderB3Delay(IN:= NOT X6D AND NOT XC3,
											PT:=T#10s,
											Q:= H2200SudsecitonCylinderB3IO.xUnload,
											ET:=m_tCylinderB3DelayCurrentTime);
IF X6D THEN
	H2200SudsecitonCylinderB3IO.xUnload:=0;
END_IF;*)(*******气缸还没装先屏蔽这段******)


(*IF NOT X3A AND NOT X3B THEN*)
m_tonSudsecitonCylinderB4Delay(IN:= NOT X6D AND NOT XC3,
											PT:=T#10s,
											Q:= H2200SudsecitonCylinderB4IO.xUnload,
											ET:=m_tCylinderB4DelayCurrentTime);
IF X6D THEN
	(*ELSIF X3A THEN*)
	H2200SudsecitonCylinderB4IO.xUnload:=0;
END_IF;

m_tonSudsecitonCylinderB5Delay(IN:= NOT X3C AND NOT X3D,
											PT:=T#10s,
											Q:= H2200SudsecitonCylinderB5IO.xUnload,
											ET:=m_tCylinderB5DelayCurrentTime);
IF X3C THEN
	H2200SudsecitonCylinderB5IO.xUnload:=0;
END_IF;

IF  X40 AND  X3F THEN
	BlockB:=1;
	ELSIF NOT X40 THEN
	BlockB:=0;
END_IF;
 
 
 


IF g_xManual OR  g_xReset THEN
	D3345:=0;
	D3350:=0;
	D3355:=0;
	D201.0:=0;
	D201.1:=0;
	D201.2:=0;
	m_xRotor1Start:=0;
	m_xRotor2Start:=0;
	m_xRotor1Done:=0;
	m_xRotor2Done:=0;
	Lifter3IO.xMDIExe:=0;
	Lifter4IO.xMDIExe:=0;
	Lifter5IO.xMDIExe:=0;
	Conveyor3IO.xLoad:=0;
	Conveyor3IO.xUnload:=0;
	Conveyor4IO.xLoad:=0;
	Conveyor4IO.xUnload:=0;
	Conveyor5IO.xLoad:=0;
	Conveyor5IO.xUnload:=0;	
	ShuttleCar1IO.xMDIExe:=0;
	ConveyorShuttleCarIO.xLoad:=0;
	ConveyorShuttleCarIO.xUnload:=0;
END_IF;
END_PROGRAM

FUNCTION_BLOCK ShuttleCar
VAR_IN_OUT
  ShuttleCarInOut : ShuttleCarIO;
END_VAR
VAR
  m_tonBrakeDelay : TON;  (* 延时 *)
  m_tBrakeDelayCurrentTime : TIME;
  m_tonArriveDelay : TON;  (* 到达延时计时器 *)
  m_xArriveDelay : BOOL;  (* 到达延时 *)
  m_tArriveDelayCurrentTime : TIME;  (* 到达延时当前时间 *)
  m_xInit : BOOL;  (* 初始化标志位 *)
  m_tonPauseDelay : TON;  (* 暂停减速 *)
  m_tPauseDelayCurrentTime : TIME;  (* 暂停延时当前时间 *)
  m_tonOvertimeAlarm : TON;  (* 超时报警定时器 *)
  m_tOvertimeCurrentTime : TIME;  (* 超时报警当前时间 *)
END_VAR
(*******************************************************************
输送小车程序，可用于使用认址片控制位置的输送车程序，可用于控制提升机，
使用了限位捕捉程序防止小车惯性过大冲过限位后继续行走，捕捉程序采用反
转复位，这样设计有弊端可能反转复位后车的位置并没有回到限位以内,当两个
限位同时碰到的时候，会使运料小车进入死锁状态，通过xPassLimit来解开死锁，
可以在触摸屏中使用一个带权限的按钮来进行控制，配合ShuttleCarCurrentPos
函数来计算位置信息
增加自动开始后将当前位置置为零的信号防止设备停在两个位置开关的中间
修改信息  修改后请增加版本
2018-1-22增加到位延时：到位延时时间可以设置，适应双向到位的位置开关，通过调整延时时间让穿梭车停在到位开关的中间
增加气缸控制信号
增加抱闸延时
增加超时报警
YAO      V1.0
2018-1-22 YAO V1.1
********************************************************************)
IF NOT m_xInit THEN
	ShuttleCarInOut.tArriveDelay:=T#0s;   (*到位延时初始化为0*)
	ShuttleCarInOut.tBrakeDelay:=T#100ms;(*抱闸延时初始化为100ms*)
	ShuttleCarInOut.tSetOverTime:=T#60s;(*超时报警初始化为1分钟*)
	m_xInit:=1;
END_IF;
(*如果是气缸的话屏蔽限位和Ready信号*)
IF ShuttleCarInOut.xCylinder THEN
	ShuttleCarInOut.xPosLimit:=1;
	ShuttleCarInOut.xNegLimit:=1;
	ShuttleCarInOut.xReady:=1;
END_IF;
(*限位捕捉，防止冲过限位开关，反转后复位*)
ShuttleCarInOut.xPosLimitCatch:=LDF(TRUE,ShuttleCarInOut.xPosLimit) OR ShuttleCarInOut.xPosLimitCatch;
IF ShuttleCarInOut.xCCW THEN  
	ShuttleCarInOut.xPosLimitCatch:=0;
END_IF;

ShuttleCarInOut.xNegLimitCatch:=LDF(TRUE,ShuttleCarInOut.xNegLimit) OR ShuttleCarInOut.xNegLimitCatch;
(*松绳报警*)
IF LDP(TRUE,ShuttleCarInOut.xLooseDetect) THEN	
	ShuttleCarInOut.xLooseAlarm:=1;
END_IF;
(*提升复位报警*)
IF ShuttleCarInOut.xCW AND NOT  ShuttleCarInOut.xLooseDetect THEN   
	ShuttleCarInOut.xLooseAlarm:=0; 
END_IF;

IF ShuttleCarInOut.xCW THEN   
	ShuttleCarInOut.xNegLimitCatch:=0; 
END_IF;

IF ShuttleCarInOut.xPassLimit OR
	g_xReset OR   (*增加复位按钮*)
	(ShuttleCarInOut.xNegLimitCatch 
	AND ShuttleCarInOut.xPosLimitCatch)  THEN  
	ShuttleCarInOut.xNegLimitCatch:=0; 
	ShuttleCarInOut.xPosLimitCatch:=0;
	ShuttleCarInOut.xLooseAlarm:=0;
END_IF;
IF ShuttleCarInOut.xReady AND g_xEStop THEN
(*手动*)
    IF g_xManual THEN  
	    IF ShuttleCarInOut.xForward 
			AND ShuttleCarInOut.xBackward=0 
			AND ShuttleCarInOut.xCCW=0 
			AND ShuttleCarInOut.xPosLimitCatch=0  THEN
		    ShuttleCarInOut.xCW:=1;
		    ELSE
		    ShuttleCarInOut.xCW:=0;
	    END_IF;
	    IF ShuttleCarInOut.xBackward 
			AND ShuttleCarInOut.xForward=0 
			AND ShuttleCarInOut.xCW=0 
			AND ShuttleCarInOut.xNegLimitCatch=0 
			AND ShuttleCarInOut.xLooseAlarm=0
			AND G_xEStop THEN  
		    ShuttleCarInOut.xCCW:=1;
		    ELSE
		    ShuttleCarInOut.xCCW:=0;
	    END_IF;
    END_IF;
    (**********)
(*自动*)
  IF g_xAuto  THEN  
  	(*点动*)
 		IF LDP(TRUE,ShuttleCarInOut.xForward) THEN
 			ShuttleCarInOut.xMDIExe:=1;
			ShuttleCarInOut.iDestinationPos:=ShuttleCarInOut.iCurrentPos+1;
		END_IF;
		IF LDP(TRUE,ShuttleCarInOut.xBackward) THEN
			ShuttleCarInOut.xMDIExe:=1;
			ShuttleCarInOut.iDestinationPos:=ShuttleCarInOut.iCurrentPos-1;
		END_IF;	 
	(*>>>>>>>>>>>>>>>>>>>>>>>>>>>>>>>>>>>>>*)	
	  IF ShuttleCarInOut.xMDIExe AND ShuttleCarInOut.iDestinationPos<>0 THEN	
	    IF ShuttleCarInOut.iCurrentPos<ShuttleCarInOut.iDestinationPos AND ShuttleCarInOut.xPosLimitCatch=0 THEN   (*正转*)
			ShuttleCarInOut.xCW:=1;
			ShuttleCarInOut.xCCW:=0;
			ShuttleCarInOut.xMDIDone:=0;
		END_IF;

		IF ShuttleCarInOut.iCurrentPos>ShuttleCarInOut.iDestinationPos AND ShuttleCarInOut.xNegLimitCatch=0 AND ShuttleCarInOut.xLooseAlarm=0 THEN   (*反转*)
			ShuttleCarInOut.xCCW:=1;
			ShuttleCarInOut.xCW:=0;
			ShuttleCarInOut.xMDIDone:=0;
		END_IF;
	m_tonArriveDelay(IN:= ShuttleCarInOut.iCurrentPos=ShuttleCarInOut.iDestinationPos ,
	                                    PT:= ShuttleCarInOut.tArriveDelay ,
	                                    Q:= m_xArriveDelay ,
	                                    ET:= m_tArriveDelayCurrentTime);
	     (*到位延时时间可以设置，适应双向到位的位置开关，通过调整延时时间让穿梭车停在到位开关的中间*)
		IF m_xArriveDelay AND NOT ShuttleCarInOut.xCylinder THEN
			ShuttleCarInOut.xCW:=0;
			ShuttleCarInOut.xCCW:=0;
			ShuttleCarInOut.xMDIDone:=1;
			ELSE
			ShuttleCarInOut.xMDIDone:=0;
		END_IF;

		IF ShuttleCarInOut.xPosLimitCatch THEN
			ShuttleCarInOut.xCW:=0;
			ShuttleCarInOut.xMDIDone:=0;
		END_IF;

		IF ShuttleCarInOut.xNegLimitCatch THEN
			ShuttleCarInOut.xCCW:=0;
			ShuttleCarInOut.xMDIDone:=0;
		END_IF;
		ELSE
		ShuttleCarInOut.xCW:=0;
		ShuttleCarInOut.xCCW:=0;
		ShuttleCarInOut.xMDIDone:=0;
	  END_IF;
	END_IF;
	ELSE  (*无就绪信号   或急停的情况下*)
		ShuttleCarInOut.xCW:=0;
		ShuttleCarInOut.xCCW:=0;	
END_IF;
    (*抱闸延时*)
m_tonBrakeDelay(IN:= ShuttleCarInOut.xCW OR ShuttleCarInOut.xCCW,
                                    PT:= ShuttleCarInOut.tBrakeDelay,
                                    Q:=ShuttleCarInOut.xBrake ,
                                    ET:= m_tBrakeDelayCurrentTime);

(*自动上电后把当前位置清零，防止穿梭车不在开关位置*)
IF LDP(TRUE,g_xAuto) THEN
	ShuttleCarInOut.iCurrentPos:=0;
END_IF;
IF ShuttleCarInOut.xCW OR ShuttleCarInOut.xCCW THEN
	ShuttleCarInOut.xBusy:=1;
	ELSE
	ShuttleCarInout.xBusy:=0;
END_IF;

(*暂停，带延时减速斜坡，ShuttleCarInOut.xPauseRamp为减速斜坡输出位*)
m_tonPauseDelay(IN:=g_xPause,PT:= T#2s ,Q:=ShuttleCarInOut.xPauseRamp,ET:= m_tPauseDelayCurrentTime );
IF ShuttleCarInOut.xPauseRamp THEN
	ShuttleCarInOut.xCW:=0;
	ShuttleCarInOut.xCCW:=0;
	ShuttleCarInOut.xBrake:=0;
END_IF;
(*超时报警*)
m_tonOvertimeAlarm(IN:= ShuttleCarInOut.xMDIExe AND (ShuttleCarInOut.iCurrentPos<>ShuttleCarInOut.iDestinationPos) ,
                                           PT:= ShuttleCarInOut.tSetOverTime,
                                           Q:= ShuttleCarInOut.xOvertimeAlarm ,
                                           ET:= m_tOvertimeCurrentTime );
END_FUNCTION_BLOCK

FUNCTION ShuttleCarCurrentPosition
VAR_INPUT
  xPosition1 : BOOL;
  xPosition2 : BOOL;
  xPosition3 : BOOL;
END_VAR
(************************************
计算输送车当前位置的函数
**************************************)
IF xPosition1 THEN
	ShuttleCarCurrentPosition:=1;
END_IF;
IF xPosition2 THEN
	ShuttleCarCurrentPosition:=2;
END_IF;
IF xPosition3 THEN
	ShuttleCarCurrentPosition:=3;
END_IF;
END_FUNCTION

FUNCTION_BLOCK ShuttleCarVelocityFB
VAR_INPUT
  xEnable : BOOL;  (* 使能 *)
  xMotorCW : BOOL;  (* 电机正转 *)
  xMotorCCW : BOOL;  (* 电机反转 *)
  xPosition1Switch : BOOL;  (* 位置1开关 *)
  xDecelerationSwitch : BOOL;  (* 减速开关 *)
  xPosition2Switch : BOOL;  (* 位置2开关 *)
END_VAR
VAR
  iFloor : INT;  (* 层数 *)
END_VAR
VAR_OUTPUT
  xHighSpeed : BOOL;
END_VAR
IF xEnable THEN
	(*电机旋转，并且在位置开关上的时候触发加速*)
	IF( LDP(TRUE,xMotorCW) AND xPosition1Switch ) OR (  LDP(TRUE,xMotorCCW) AND xPosition2Switch) THEN
		xHighSpeed:=1;
		iFloor:=0;
	END_IF;
	IF LDF(TRUE,xMotorCW) OR LDF(TRUE,xMotorCCW) THEN
		xHighSpeed:=0;
    END_IF;
	IF LDP(TRUE,xDecelerationSwitch) THEN
		iFloor:=iFloor+1;
	END_IF;
	IF iFloor=2 THEN
		xHighSpeed:=0;
		iFloor:=0;
	END_IF;
ELSE
    xHighSpeed:=0;
END_IF;
END_FUNCTION_BLOCK

PROGRAM Start
IF g_xReset THEN
	SM50:=1;
ELSE
	SM50:=0;
END_IF;
CASE g_iState OF
	0: 
		g_xManual:=1;
		g_xAuto:=0;	
		g_xStackLampAmber:=1;
		g_xStackLampGreen:=0;
		g_xRemoteAuto:=0;
	1:
		g_xManual:=0;
		g_xAuto:=1;
		g_xStackLampGreen:=1;
		g_xStackLampAmber:=0;
		g_xRemoteAuto:=0;
	2:	
        g_xRemoteAuto:=1;
        g_xStackLampGreen:=1;
        g_xStackLampAmber:=0;
        g_xAuto:=0;
		g_xManual:=0;
END_CASE;
IF g_xLocalAutoStart THEN  
	g_iState:=1;
END_IF;
IF g_xAlarm  AND SM412 THEN
	g_xStackLampRed:=1;
	g_xBuzzer:=1;
ELSE
	g_xStackLampRed:=0;
	g_xBuzzer:=0;	
END_IF;
IF g_xStop OR g_xEStop=0 THEN 
	g_iState:=0;
END_IF;
IF g_xRemoteAutoStart THEN
	g_iState:=2;
END_IF;
IF g_xPause AND SM412 THEN
	g_xStackLampGreen:=0;
	g_xStackLampAmber:=0;
END_IF;
END_PROGRAM

PROGRAM UDP
VAR
  m_ton4ReceiveHeartbeat : TON;  (* 心跳信号接收上升沿 *)
  m_t4RecHeartbeatCurrentTime : TIME;  (* 心跳信号接收当前时间 *)
  m_ton5ReceiveHeartbeat : TON;  (* 心跳信号接收上升沿 *)
  m_t5RecHeartbeatCurrentTime : TIME;  (* 心跳信号接收当前时间 *)
  m_ton1ReceiveHeartbeat : TON;  (* 心跳信号接收上升沿 *)
  m_t1RecHeartbeatCurrentTime : TIME;  (* 心跳信号接收当前时间 *)
  m_ton2ReceiveHeartbeat : TON;  (* 心跳信号接收上升沿 *)
  m_t2RecHeartbeatCurrentTime : TIME;  (* 心跳信号接收当前时间 *)
  m_ton1ReceiveReConnect : TON;
  m_ton2ReceiveReConnect : TON;
  m_ton4ReceiveReConnect : TON;
  m_ton5ReceiveReConnect : TON;
  m_x1ReceiveReConnect : BOOL;
  m_x2ReceiveReConnect : BOOL;
  m_x4ReceiveReConnect : BOOL;
  m_x5ReceiveReConnect : BOOL;
  m_t1ReceiveReConnectCurrentTime : TIME;
  m_t2ReceiveReConnectCurrentTime : TIME;
  m_t4ReceiveReConnectCurrentTime : TIME;
  m_t5ReceiveReConnectCurrentTime : TIME;
END_VAR
(*化成1号柜TCP通讯*)
D200:=k2;
D332:=1;
D333:=2;
SP_SOCRMODE(LDP(TRUE,SM402), "U0" , K1 , D330 );
SP_SOCCINF( LDP(TRUE,SD1282.0) , "U0" , K1 , D110 ,D120);
SP_SOCSND( SM412 AND SD1282.0 , "U0" , K1 , D100, D200, M102 );
SP_SOCRCV(NOT M104 AND SD1282.0  ,
							 "U0" , 
							 K1,               
							 D300 , 
							 D400 ,
							 M104 );
D201.F:=SM413;
m_ton1ReceiveHeartbeat(IN:=NOT LDP(TRUE, D401.F) ,PT:= t#5S ,Q:= g_xChem1ComFailed ,ET:= m_t1RecHeartbeatCurrentTime);
IF g_xChem1ComFailed THEN
	D400:=0;
	D401:=0;
	M104:=SM413;(*通讯失败有可能是接收模块没动作，重启接收模块*)
END_IF;
(*化成RGV，TCP通讯*)
D220:=k10;
SP_SOCCINF( LDP(TRUE,SD1282.3) , "U0" , K4 , D140 ,D150);
SP_SOCSND( SM412 AND SD1282.3 , "U0" , K4 , D160, D220, M106 );
SP_SOCRCV( NOT M108  AND SD1282.3 , "U0" , K4, D310 , D420 ,M108 );
D223.F:=SM413;
m_ton4ReceiveHeartbeat(IN:=NOT LDP(TRUE, D422.F) ,PT:= t#5S ,Q:= g_xChemRGVComFailed ,ET:= m_t4RecHeartbeatCurrentTime);

IF  g_xChemRGVComFailed  THEN
	M108:=SM413;(*通讯失败有可能是接收模块没动作，重启接收模块*)
	D420:=0;
	D421:=0;
	D422:=0;
	D423:=0;
	D424:=0;
END_IF;
(*二封RGV，TCP通讯*)
D240:=k22;
SP_SOCCINF( LDP(TRUE,SD1282.4) , "U0" , K5 , D170 ,D180);
SP_SOCSND( SM412 AND SD1282.4 , "U0" , K5 , D190, D240, M110);
SP_SOCRCV( NOT M112 AND SD1282.4 , "U0" , K5, D320 , D430 ,M112 );
D243.F:=SM413;
m_ton5ReceiveHeartbeat(IN:=NOT LDP(TRUE, D433.F) ,PT:= t#5S ,Q:= g_xQuarPackageRGVComFailed ,ET:= m_t5RecHeartbeatCurrentTime);

IF  g_xQuarPackageRGVComFailed THEN
	M112:=SM413;(*通讯失败有可能是接收模块没动作，重启接收模块*)
	D430:=0;
	D431:=0;
	D432:=0;
	D433:=0;
	D434:=0;
END_IF;
END_PROGRAM

FUNCTION_BLOCK AccumulateConveyor
VAR_IN_OUT
  AccumulateConveyorIO : AccumulateConveyorIO;
END_VAR
VAR
  m_tpViaDelay : TP;  (* 卸料延时定时器 *)
  m_xViaDelay : BOOL;  (* 通过延时 *)
  m_tViaDelayElapse : TIME;  (* 通过延时当前时间 *)
  m_xInitial : BOOL;  (* 初始化 *)
  m_xOccupy : BOOL;
  m_tonUnloadDelay : TON;
  m_xUnloadDelay : BOOL;
  m_tUnloadDelay : TIME;
  m_tpOcuppyDelay : TP;
  m_xOccupy2 : BOOL;
  iStep : INT;
  m_tonLoadDelay : TON;  (* 上料延时 *)
  m_xLoadDelay : BOOL;
  m_tLoadDelay : TIME;
  m_xLoading : BOOL;  (* 上料中 *)
  m_xUnloading : BOOL;  (* 下料中 *)
  m_tonDischargeDelay : TON;
  m_xDischargeDelay : BOOL;  (* 上料中 *)
  m_tDischargeDelay : TIME;  (* 下料中 *)
END_VAR
  (***********************************************************************
阻挡器模块，
由一个行程开关，一个阻挡器，一个倍速链输送电机组成
具有手动与自动模式
xEmpty显示当前为空料的状态
xUnload为卸料信号，连接下一设备的xEmpty信号
*************************************************************************)

  (*初始化，离开延时时间设置为5秒*)
IF NOT m_xInitial THEN
	 AccumulateConveyorIO.tLeaveDelay :=T#3s;
	 AccumulateConveyorIO.tLoadDelay:=T#3S;
	m_xInitial:=1;
END_IF;
IF g_xManual THEN    (*手动*)
	AccumulateConveyorIO.xNextRun:=0;
	AccumulateConveyorIO.xBarCylinder:=AccumulateConveyorIO.xBarCylinderButton;
	AccumulateConveyorIO.xTransportMotorCW:=AccumulateConveyorIO.xTransportMotorCWButton 
																						AND NOT AccumulateConveyorIO.xTransportMotorCCWButton 
																						AND NOT AccumulateConveyorIO.xTransportMotorCCW;
	AccumulateConveyorIO.xTransportMotorCCW:=AccumulateConveyorIO.xTransportMotorCCWButton 
																							AND NOT AccumulateConveyorIO.xTransportMotorCWButton 
																							AND NOT AccumulateConveyorIO.xTransportMotorCW;
END_IF;
(*离开延时定时器*)
m_tpViaDelay(IN:=LDF(TRUE,AccumulateConveyorIO.xPresentSwitchEntry)  AND AccumulateConveyorIO.xLoad  AND g_xAuto  ,
						PT:= AccumulateConveyorIO.tLeaveDelay ,
						Q:= m_xOccupy ,
						ET:=m_tViaDelayElapse );
m_tpOcuppyDelay(IN:= LDF(TRUE,m_xOccupy) ,PT:= t#2S,Q:= m_xOccupy2  ,ET:=m_tViaDelayElapse );						
 AccumulateConveyorIO.xEmpty:=NOT m_xOccupy2;
m_tonUnloadDelay(IN:= AccumulateConveyorIO.xUnload AND AccumulateConveyorIO.xPresentSwitchEntry AND g_xAuto ,
     								PT:= T#3s ,(*下料时，如果东西不在阻挡的位置，往前转，转到阻挡被挡住一段时间再卡住第二个*)
     								Q:= m_xUnloadDelay ,
     								ET:=m_tUnloadDelay);
m_tonLoadDelay(IN:=iStep=3,(*上料延时，上料检测到东西后，多转一会儿，转过阻挡，防止顶起来顶到框*)
											PT:=AccumulateConveyorIO.tLoadDelay,
											Q:=m_xLoadDelay,
											ET:=m_tLoadDelay);
m_tonDischargeDelay(IN:=iStep=4,(*下料完毕，多运转一会儿，把第二个框放过去，也可以改为0，因为unload延时也有这个效果*)
											PT:=T#3S,
											Q:=m_xDischargeDelay,
											ET:=m_tDischargeDelay);   								
(*IF LDF(TRUE,AccumulateConveyorIO.xPresentSwitchEntry) AND AccumulateConveyorIO.xLoad THEN
	AccumulateConveyorIO.iAccumulate:=AccumulateConveyorIO.iAccumulate+1;
END_IF;
IF LDF(TRUE,AccumulateConveyorIO.xPresentSwitchEntry) AND AccumulateConveyorIO.xUnload THEN
	AccumulateConveyorIO.iAccumulate:=AccumulateConveyorIO.iAccumulate-1;
END_IF;*)
IF g_xAuto THEN(*自动*)
	CASE iStep OF
		0:
		AccumulateConveyorIO.xTransportMotorCW:=0;
   	    AccumulateConveyorIO.xTransportMotorCCW:=0;
   	    AccumulateConveyorIO.xBarCylinder:=0;	
   	    AccumulateConveyorIO.xBarCylinderSecondary:=0;
   	   	AccumulateConveyorIO.xNextRun:=0;
   	   	AccumulateConveyorIO.xLoadDone:=0;
		IF g_xEStop THEN
			IF AccumulateConveyorIO.xLoad OR m_xLoading THEN 
				istep:=1;
				ELSIF AccumulateConveyorIO.xUnload AND AccumulateConveyorIO.iAccumulate>0 OR m_xUnloading THEN 
				iStep:=2;
			END_IF;	
		END_IF;		
		1:
		m_xLoading:=1;
		IF AccumulateConveyorIO.xTwoWay THEN 
			AccumulateConveyorIO.xTransportMotorCW:=0;
	   	   AccumulateConveyorIO.xTransportMotorCCW:=1;	   
	   	   AccumulateConveyorIO.xBarCylinder:=1;	  
	   	   AccumulateConveyorIO.xBarCylinderSecondary:=0;  
		ELSE
			AccumulateConveyorIO.xTransportMotorCW:=1;
	   	   AccumulateConveyorIO.xTransportMotorCCW:=0;	   
	   	   AccumulateConveyorIO.xBarCylinder:=0;	  
	   	   AccumulateConveyorIO.xBarCylinderSecondary:=0;  			
	   END_IF;
			IF LDP(TRUE,AccumulateConveyorIO.xPresentSwitchEntry) AND AccumulateConveyorIO.xTwoWay(*反向上料，检测到阻挡处的行程停*)
				OR LDP(TRUE,AccumulateConveyorIO.xPresentSwitch)AND NOT AccumulateConveyorIO.xTwoWay THEN (*正向上料，检测到尾端行程停*)
				AccumulateConveyorIO.xLoadDone:=1; 
				AccumulateConveyorIO.iAccumulate:=AccumulateConveyorIO.iAccumulate+1;
		    	iStep:=3;
			END_IF;
		2:
		m_xUnloading:=1;
		AccumulateConveyorIO.xNextRun:=1;
		AccumulateConveyorIO.xTransportMotorCW:=1;
    	AccumulateConveyorIO.xTransportMotorCCW:=0;
        IF m_xUnloadDelay   THEN
    	AccumulateConveyorIO.xBarCylinder:=1;
    	AccumulateConveyorIO.xBarCylinderSecondary:=1;
   		END_IF;
  		IF NOT  AccumulateConveyorIO.xUnload  THEN
    		AccumulateConveyorIO.iAccumulate:=AccumulateConveyorIO.iAccumulate-1;
    		iStep:=4;
  		END_IF;
		3:(*开关检测到再多走一会儿，免得顶起时撞到框*)
		m_xLoading:=0;

		IF m_xLoadDelay THEN
			iStep:=0;
		END_IF;	
		4:(*unload完,一般都是下段not empty了，把下一个放出来*)
		m_xUnloading:=0;
		AccumulateConveyorIO.xBarCylinder:=0;
		AccumulateConveyorIO.xBarCylinderSecondary:=0;

		IF m_xDischargeDelay THEN
			iStep:=0;
		END_IF;	
	END_CASE;		
END_IF;
 (*   IF AccumulateConveyorIO.xUnload  AND AccumulateConveyorIO.iAccumulate>0 AND NOT AccumulateConveyorIO.xNextRun THEN(*收到卸料命令，当阻挡器不为空时*)   	  
 (*	AccumulateConveyorIO.xNextRun:=1;(*确保下料命令只执行一次，防止物料在输送过程中又有卸料命令导致多事卸料*)
 (*	AccumulateConveyorIO.xTransportMotorCW:=1;
    	AccumulateConveyorIO.xTransportMotorCCW:=0;
    END_IF;
    IF m_xDischargeDelay   THEN
    	AccumulateConveyorIO.xBarCylinder:=1;
    	AccumulateConveyorIO.xBarCylinderSecondary:=1;
    END_IF;
    IF NOT  AccumulateConveyorIO.xUnload  THEN
    	AccumulateConveyorIO.xNextRun:=0;
    END_IF;*)
    (*如果为空，气缸顶起*)
   (*  IF AccumulateConveyorIO.xLoad AND NOT AccumulateConveyorIO.xTwoWay AND NOT AccumulateConveyorIO.xUnload THEN
	   	   AccumulateConveyorIO.xTransportMotorCW:=1;
	   	   AccumulateConveyorIO.xTransportMotorCCW:=0;	 
	   	   AccumulateConveyorIO.xBarCylinder:=1;	 
	   	   AccumulateConveyorIO.xBarCylinderSecondary:=0;  	   
		ELSIF AccumulateConveyorIO.xLoad AND AccumulateConveyorIO.xTwoWay  AND NOT AccumulateConveyorIO.xUnload THEN
	   	   AccumulateConveyorIO.xTransportMotorCW:=0;
	   	   AccumulateConveyorIO.xTransportMotorCCW:=1;	   
	   	   AccumulateConveyorIO.xBarCylinder:=1;	  
	   	   AccumulateConveyorIO.xBarCylinderSecondary:=0;  
	   END_IF;

  IF NOT AccumulateConveyorIO.xUnload AND NOT  AccumulateConveyorIO.xLoad THEN
   	    AccumulateConveyorIO.xTransportMotorCW:=0;
   	    AccumulateConveyorIO.xTransportMotorCCW:=0;
   	    AccumulateConveyorIO.xBarCylinder:=0;	
   	    AccumulateConveyorIO.xBarCylinderSecondary:=0;
   	END_IF;
END_IF;*)
IF NOT g_xEStop THEN
	AccumulateConveyorIO.xTransportMotorCW:=0;
	 AccumulateConveyorIO.xTransportMotorCCW:=0;
	 AccumulateConveyorIO.xBarCylinder:=0;
END_IF;
(*插入数量*)
IF g_xInsertTask AND AccumulateConveyorIO.iDeviceID=g_iDeviceIDSelect THEN
	AccumulateConveyorIO.iAccumulate:=g_iInsertTask;
END_IF;	
(*复位*)
IF (g_xResetSingle AND AccumulateConveyorIO.iDeviceID=g_iDeviceIDSelect)THEN
	iStep:=0;
	m_xLoading:=0;
	m_xUnloading:=0;
END_IF;
END_FUNCTION_BLOCK

FUNCTION_BLOCK PriorityFB
VAR_INPUT
  arrxCondition : ARRAY [0..9] OF BOOL;
  xTaskComplete : BOOL;  (* 任务完成 *)
  xReset : BOOL;  (* 复位 *)
END_VAR
VAR
  xOccupy : BOOL;  (* 占用 *)
END_VAR
VAR_OUTPUT
  iPriority : INT;  (* 输出任务号 *)
END_VAR
VAR
  jj : INT;
END_VAR
VAR CONSTANT
  CONDITION_QUANTITY : INT := 10;
END_VAR
VAR
  arriTaskStack : ARRAY [0..10] OF INT;
  ii : INT;
  kk : INT;
  arrtConditionDelay : ARRAY [0..9] OF TIME := [10(T#0s)];
  arrxConditionEdgeDetect : ARRAY [0..9] OF BOOL;
END_VAR
(****************************************************************************)
(*
优先级功能块，存储5个条件的优先级，实现栈功能先入先出，
复位功能还有问题，
出入栈式优先级块，满足条件后入栈，先入先出，在栈尾加载新任务
栈首为当前执行的任务，任务完成使用上升沿触发，触发后栈首元素弹出

复位功能清空堆栈，栈的容量在CONDITION_QUANTITY 设置
*)

(***************************************************************************)
(*入栈
//out_t(arrxCondition[1],arrtConditionDelay[1],20);*)
FOR ii:=1 TO CONDITION_QUANTITY BY 1 DO	
	IF arrxCondition[ii] AND NOT arrxConditionEdgeDetect[ii] THEN;
		FOR kk:=0 TO CONDITION_QUANTITY BY 1 DO
			IF arriTaskStack[kk]=0 THEN
				arriTaskStack[kk]:=ii;
				EXIT;
			END_IF;		
		END_FOR;
	END_IF;	
	arrxConditionEdgeDetect[ii]:=arrxCondition[ii];
END_FOR;
(*栈顶任务为当前执行的任务*)
iPriority:=arriTaskStack[0];
(*栈顶任务完成，弹出*)
IF 	LDP(TRUE, xTaskComplete) THEN
	FOR jj:=0 TO CONDITION_QUANTITY-1 BY 1 DO
		arriTaskStack[jj]:=arriTaskStack[jj+1];
	END_FOR;
	arriTaskStack[CONDITION_QUANTITY]:=0;
END_IF;
(*复位*)
IF LDP(TRUE,xReset) THEN
	FOR jj:=0 TO CONDITION_QUANTITY BY 1 DO
		arriTaskStack[jj]:=0;
	END_FOR;
	FOR jj:=1 TO CONDITION_QUANTITY BY 1 DO
		arrxConditionEdgeDetect[jj]:=0;
	END_FOR;
END_IF;
END_FUNCTION_BLOCK
